// SIMATIC S7-200 project (STEP 7-Micro/WIN), CPU 226 REL 02.01

SYMBOL_TABLE 用户定义1
TS_IndexMotor    V1001.0
TS_ResetButton   V1000.0
Station_Alarm    V107.6
S6_Alarm         V168.7
S5_Alarm         V158.7
S4_Alarm         V148.7
S3_Alarm         V138.7
HomeApprop       M5.7
WaitStart        V3101.0
Running          V3101.1
Initilizing      V3100.1
WaitIni          V3100.0
TS_Rset_3D_0     V2000.7
TS_Rset_3C_0     V2000.5
TS_Rset_3B0      V2000.3
E_Stop           M0.0
Start_Button     M0.1
Stop_Button      M0.2
Reset_Button     M0.3
Bypass           M0.4
Safety_Relay     M0.5
MW_Switch        M0.6
Safety_Curtain   M0.7
S1_Ball_Screw    M1.0
S1_OE1           M1.1
S1_OE2           M1.2
S1_OE3           M1.3
S1_Cover_Group   M1.4
S1_Color         M1.5
S1_ORing         M1.6
SpareM1_7        M1.7
S2Ball_Screw     M2.0
S2OE21           M2.1
S2OE2            M2.2
S2OE3            M2.3
S2_Cover_Group   M2.4
Color_Sensor     M2.5
S2ORing          M2.6
Cyl3A_S0         M3.0
Cyl3A_S1         M3.1
Cyl3B_S0         M3.2
Cyl3B_S1         M3.3
Cy3C_S1          M3.5
Cyl3C_S0         M3.4
Cyl3D_S0         M3.6
CyL3D_S1         M3.7
Cyl_4A_S0        M4.0
Cyl4A_S1         M4.1
Cyl4B_S0         M4.2
Cyl4B_S1         M4.3
Cyl4C_S0         M4.4
Cyl4C_S1         M4.5
Cyl4D_S0         M4.6
Cyl4D_S1         M4.7
Laser_Marking    M5.0
Laser_done       M5.1
Cyl6A_S0         M6.0
Cyl6A_S1         M6.1
Cyl6B_S0         M6.2
Cyl6B_S1         M6.3
Cyl6C_S0         M6.4
Cyl6C_S1         M6.5
SpareM6_6        M6.6
SpareM6_7        M6.7
ServoMotorBLimit M7.0
Servo_Home_Pos   M7.1
ServoMotorFLimit M7.2
ServoAlarm       M7.3
ServoReady       M7.4
Cyl3E_S0         M8.0
Cyl3E_S1         M8.1
Cyl3F_S0         M8.2
Cyl3F_S1         M8.3
SpareM8_4        M8.4
SpareM8_5        M8.5
Cyl2A_S0         M8.6
Cyl2A_S1         M8.7
IndexOrig_Pos    M9.0
Reject_Box_1     M9.1
Reject_Box_2     M9.2
Reject_Box_3     M9.3
Reject_Box_4     M9.4
PC_Test_Complete_1 M9.5
PC_Test_Complete_2 M9.6
SafetyDoor       M9.7
CurrentTestOK_1  M10.0
CurrentTestNG_1  M10.1
RunTimeTestOK_1  M10.2
RunTimeTestNG_1  M10.3
LeakageTestOK_1  M10.4
LeakageTestNG_1  M10.5
LeakageTestAlarm_1 M10.6
Add_10N_Force_1  M10.7
CurrentTestOK_2  M11.0
CurrentTestNG_2  M11.1
RunTimeTestOK_2  M11.2
RunTimeTestNG_2  M11.3
LeakageTestOK_2  M11.4
LeakageTestNG_2  M11.5
LeakageTestAlarm_2 M11.6
Add_10N_Force_2  M11.7
CW               M20.0
CCW              M20.1
ServoEnable      M20.2
DelServoAlarm    M20.3
Up_Down_Cyl_1    M20.4
Up_Down_Cyl_2    M20.5
Pic_Product_Cyl_1 M20.6
Pic_Product_Cyl_2 M20.7
TW_G             M21.0
TW_R             M21.1
TW_Buzzer        M21.2
Reset_lamp       M21.3
Bypass_Lamp      M21.4
SV_3E_0          M22.0
SV_3E_1          M22.1
SV_3F_0          M22.2
SV_3F_1          M22.3
EnableTest_to_PC1 M22.4
EnableTest_to_PC2 M22.5
SV_3A_0          M23.0
SV_3A_1          M23.1
SV_3B_0          M23.2
SV_3B_1          M23.3
SV_3C_0          M23.4
SV_3C_1          M23.5
SV_3D_0          M23.6
SV_3D_1          M23.7
SV_4A_0          M24.0
SV_4A_1          M24.1
SV_4B_2mmCYL     M24.2
SV_4C_RotateCyl  M24.3
SV_4D_RotateCyl  M24.4
Index_Brake      M24.5
Servo_Brake      M24.6
MainValve        M24.7
Index_Motor      M25.0
ConverMotor      M25.1
RejectBox_Cyl    M25.2
Start_Laser      M25.3
Stop_Laser       M25.4
SpareM25_5       M25.5
Alarm1_ToPC      M25.6
Alarm2_ToPC      M25.7
StartLeakage_1   M26.0
ResetLeakage_1   M26.1
Romote_Eable_1   M26.2
StartLeakage_2   M27.0
ResetLeakage_2   M27.1
Romote_Eable_2   M27.2
StationRunTag    V0.0
TurnplateRunTag  V0.1
SysIniOk         V0.5
DeviceIniOk      V0.6
Ini_OK_Tag       V0.7
StationIniStatus V1.0
Station1IniStatus V1.1
Station2IniStatus V1.2
Station3IniStatus V1.3
Station4IniStatus V1.4
Station5IniStatus V1.5
Station6IniStatus V1.6
IniTags          V1.7
TypeCheckOk      V2.1
Auto_Mode        V3.0
TW_Ini_Status    V4.0
S5_To_S6_Ok      V9.0
S4_To_S5_Ok      V9.1
S3_To_S4_Ok      V9.2
S2_To_S3_Ok      V9.3
SS_Transfer_Ok   V9.7
Start_Signal     V10.7
S2_Complete_Tag  V27.7
下行汽缸AB           V36.1
通电汽缸             V36.2
移除砝码             V36.6
移除插座             V36.7
释放产品             V37.0
S3_CompleteTag   V37.7
S4_Product_Enable_Tag_1 V40.1
S4_Product_Enable_Tag_2 V40.2
S4_ProductEnable V40.3
S4_Complete_Tag  V47.7
Sent_Ok          V50.7
S5_Complete_Tag  V57.7
Release1st_1     V60.4
Release1st_2     V60.5
S6_Complete_Tag  V67.7
Fatal_Alarm      V107.7
TS_Start         V1000.1
TS_Stop          V1000.2
TS_Reset         V1000.3
Index_Signal_Edge V1000.7
Product_set      V1999.7
TS_Set_3A        V2000.0
TS_Reset_3A      V2000.1
TS_Set_3B        V2000.2
TS_Set_3C        V2000.4
TS_Set_3D        V2000.6
TS_Set_3E        V2001.0
TS_Set_3F        V2001.2
TS_Current_Test  V2001.4
TS_Set_4A        V2004.0
TS_Reset_4A      V2004.1
Maintain_mode    V2009.7
Single_Mode      V2019.7
TS_Laser_Test    V2049.0
TS_Laser_Stop    V2049.1
END_SYMBOL_TABLE

SYMBOL_TABLE S7-200 符号
Always_On        SM0.0    // 始终接通为 ON
First_Scan_On    SM0.1    // 仅第一个扫描周期中接通为 ON
Clock_1s         SM0.5    // 在 1 秒钟的循环周期内，接通为 ON 0.5 秒，关断为 OFF 0.5  秒
PLS0_Enable      SM67.7   // PTO0/PWM0 使能：1 = 使能
PLS1_Enable      SM77.7   // PTO1/PWM1 使能：1 = 使能
PLS0_Ctrl        SMB67    // PTO0/PMW0 监控，用于 Q0.0 上的 PTO（脉冲串输出）和PWM（脉冲宽度调制）
PLS1_Ctrl        SMB77    // PTO1/PWM1 监控，用于 Q0.1 上的 PTO（脉冲串输出）和 PWM（脉冲宽度调制）
PTO0_PC          SMD72    // PTO0 脉冲计数值：双字整数（1至2^32 - 1）
PTO1_PC          SMD82    // PTO1 脉冲计数值：双字整数（1至2^32 - 1）
PLS0_Cycle       SMW68    // PTO0/PWM0 周期时间值：字数据类型（2 至 65,535 个时基单位）
PLS1_Cycle       SMW78    // PTO1/PWM1 周期时间值：字数据类型（2 至 65,535 个时基单位）
END_SYMBOL_TABLE

ORGANIZATION_BLOCK Main_program:OB1
TITLE=项目信息 
// 这个PLC程序控制一个6工位转盘系统，用于在汽车零部件装配线上实现自动化装配和测试，主要针对刹车阀或油泵等部件。
// 系统通过PLC管理转盘的旋转和各工位的操作，支持自动和手动模式，并在自动模式下通过运行标志V0.0置位启动转盘运行。
// 程序记录测试结果和生产数据VW2050、VW2054，用于后续生产管理和质量控制。
// 物理设备包括6工位转盘、进料机构、类型检测机构、电气测试机构、泄漏测试机构、打标机构、下料机构、传感器和执行器。
// 
// 系统流程
// 操作员通过触摸屏通信监控系统状态，并可选择自动模式或手动模式运行。按下启动按钮后，若安全条件满足，系统将置位转盘运行标志，启动转盘旋转，各工位按序执行任务。系统上电时，系统初始化确保所有硬件复位并加载参数，设备初始化完成和系统初始化完成信号确认后，生产才能开始。
// 生产流程从上料工位控制开始，零件被放置在转盘上，通过传感器检测零件到位后，上料动作完成。转盘旋转到下一工位后，类型检测工位控制通过传感器识别刹车阀型号。随后，电气测试工位控制检测电气性能，合格与否记录在生产计数器中。接着，泄漏测试工位控制检查气密性，若泄漏测试仪报警触发，系统会停止该工位操作以防止次品流出。合格零件进入打标工位控制，由激光设备刻印标识，最后通过下料工位控制卸载成品，伺服马达控制将零件送至指定位置。
// 系统在运行过程中，急停按钮用于监控设备状态，确保异常时及时干预。急停按钮被按下时，系统会立即停止所有操作，包括复位转盘运行标志，确保紧急情况下设备停机。当安全门打开时，系统将阻止转盘运行标志的置位，确保人员安全。安全继电器断电时，系统直接切断转盘电机的电源，避免电气故障。气压开关检测到气压不足时，系统暂停所有气动执行器的操作，确保动作可靠。运行中若安全光栅被遮挡，系统不置位转盘旋转标志，保护操作员安全。伺服马达报警触发时，系统禁用伺服马达使能，防止设备损坏。转盘运行标志置位前，系统需确认安全门关闭、安全继电器正常、气压充足等条件，确保运行平稳。报警处理检测到异常时，系统根据报警类型停止相关工位操作，保障安全。
// 
// 
// 【代码最后更新与2008年6月10日】
BEGIN
Network 1 // 网络标题
// 网络注释
LD     Always_On:SM0.0
CALL   Station1_Load:SBR0
?000
Network 2
LD     Always_On:SM0.0
CALL   Station2_TypeCheck:SBR1
Network 3
LD     Auto_Mode:V3.0
AN     Single_Mode:V2019.7
O      V2010.3
AN     TS_ResetButton:V1000.0
AN     Reset_Button:M0.3
AN     TS_Stop:V1000.2
CALL   Station3_E_Test:SBR2
Network 4
LD     Auto_Mode:V3.0
AN     Single_Mode:V2019.7
O      V2010.4
AN     Reset_Button:M0.3
AN     TS_ResetButton:V1000.0
AN     TS_Stop:V1000.2
CALL   Station4_L_Test:SBR3
Network 5
LDN    Single_Mode:V2019.7
O      V2010.5
AN     TS_ResetButton:V1000.0
AN     Reset_Button:M0.3
AN     TS_Stop:V1000.2
CALL   Station5_LMark:SBR4
Network 6
LD     Auto_Mode:V3.0
AN     Single_Mode:V2019.7
O      V2010.6
AN     Reset_Button:M0.3
AN     TS_ResetButton:V1000.0
AN     TS_Stop:V1000.2
CALL   Station6_Unload:SBR5
Network 7
LD     Always_On:SM0.0
CALL   Machine_alarm:SBR6
Network 8
LD     Always_On:SM0.0
CALL   Product_alarm:SBR7
Network 9
LD     Always_On:SM0.0
CALL   Ini:SBR8
Network 10
LD     Always_On:SM0.0
CALL   Turn:SBR9
Network 11
LD     Always_On:SM0.0
CALL   Servo_motor:SBR10
Network 12
LD     Always_On:SM0.0
CALL   Input:SBR11
Network 13
LD     Always_On:SM0.0
CALL   Output:SBR12
Network 14
LD     Always_On:SM0.0
CALL   TP170:SBR13
Network 15
LD     Always_On:SM0.0
CALL   Tags:SBR14
Network 16
LD     Always_On:SM0.0
CALL   PowerOn:SBR15
Network 17
LD     Always_On:SM0.0
CALL   SyS_MSG:SBR16
Network 18
LD     Always_On:SM0.0
CALL   Man_MSG:SBR17
Network 19
LD     Always_On:SM0.0
CALL   Communication_Laser:SBR18
END_ORGANIZATION_BLOCK

SUBROUTINE_BLOCK Station1_Load:SBR0
TITLE=子程序注释
BEGIN
Network 1 // 网络标题
// 网络注释
LD     Safety_Curtain:M0.7
EU
=      Start_Signal:V10.7
END_SUBROUTINE_BLOCK

SUBROUTINE_BLOCK Station2_TypeCheck:SBR1
TITLE=子程序注释
BEGIN
Network 1
// 等待启动信号
LD     IndexOrig_Pos:M9.0
EU
A      SysIniOk:V0.5
A      V26.0
A      Auto_Mode:V3.0
AN     TS_ResetButton:V1000.0
MOVB   2, VB26
Network 2
// 固定产品
LDN    TurnplateRunTag:V0.1
A      V26.1
AN     Cyl2A_S0:M8.6
A      Cyl2A_S1:M8.7
LPS
A      T33
MOVB   4, VB26
LPP
TON    T33, +50
Network 3
LDN    TurnplateRunTag:V0.1
A      V26.2
AN     Cyl2A_S1:M8.7
A      Cyl2A_S0:M8.6
MOVB   8, VB26
Network 4
// vb=6,Type=007 878-04
LDN    TurnplateRunTag:V0.1
LD     V26.3
O      Maintain_mode:V2009.7
ALD
CALL   TypeCheck:SBR19
CALL   TypeCheck1:SBR20
Network 5
LDN    TurnplateRunTag:V0.1
A      V26.3
LPS
A      T35
MOVB   16, VB26
LPP
TON    T35, +50
Network 6
// 放开产品
LDN    TurnplateRunTag:V0.1
A      V26.4
A      Cyl2A_S0:M8.6
AN     Cyl2A_S1:M8.7
MOVB   32, VB26
Network 7
LDN    TurnplateRunTag:V0.1
A      V26.5
MOVB   1, VB26
Network 8
LDB=   VB21, VB23
OB=    VB21, 0
LDB=   VB22, VB23
OB=    VB22, 0
ALD
=      TypeCheckOk:V2.1
Network 9
LDB=   VB23, 0
=      V121.6
Network 10
LDB=   VB23, 5
OB=    VB23, 6
=      M21.6
Network 11
LDB=   VB23, 1
OB=    VB23, 3
OB=    VB23, 5
=      M26.6
Network 12
LDB=   VB23, 2
OB=    VB23, 3
OB=    VB23, 6
=      M26.7
Network 13
LDB=   VB23, 4
OB=    VB23, 5
OB=    VB23, 6
=      M27.6
END_SUBROUTINE_BLOCK

SUBROUTINE_BLOCK Station3_E_Test:SBR2
TITLE=vb30--3b39;T130-----T149
BEGIN
Network 1
// 等待启动信号
LD     IndexOrig_Pos:M9.0
EU
LPS
A      V30.3
A      SysIniOk:V0.5
A      V36.0
MOVB   2, VB36
LRD
AN     V30.1
MOVB   VB31, VB33
LPP
AN     V30.2
MOVB   VB32, VB34
Network 2
// v31.1汽缸A和B下行（对应m3.1和m3.3感应信号）
LDN    TurnplateRunTag:V0.1
A      V30.3
A      下行汽缸AB:V36.1
LPS
LDN    Cyl3A_S0:M3.0
A      Cyl3A_S1:M3.1
ON     V30.1
LDN    Cyl3B_S0:M3.2
A      Cyl3B_S1:M3.3
ON     V30.2
ALD
ALD
MOVB   4, VB36
LPP
TON    T131, +20
Network 3
// V36.2 给产品通电。汽缸E为水平方向方的通电汽缸,对应产品类型为1、2、3、4；
// 汽缸F为垂直方向的通电汽缸；对应产品类型为5、6
LDN    TurnplateRunTag:V0.1
A      V30.3
A      通电汽缸:V36.2
LPS
LDB<=  VB23, 4
AN     Cyl3F_S0:M8.2
A      Cyl3F_S1:M8.3
LDB>=  VB23, 5
AN     Cyl3E_S0:M8.0
A      Cyl3E_S1:M8.1
OLD
ALD
TON    T32, +0
A      T32
MOVB   8, VB36
LPP
TON    T132, +20
Network 4 // 网络标题
// v36.3为提供给PC的测试Ready 信号，m10.7,m11.7 电流测试完成信号(也即加砝码信号，PC提供)，v36.4加砝码
LDN    TurnplateRunTag:V0.1
A      V30.3
A      V36.3
LPS
LD     EnableTest_to_PC1:M22.4
A      Add_10N_Force_1:M10.7
ON     V30.1
O      CurrentTestNG_1:M10.1
LD     EnableTest_to_PC2:M22.5
A      Add_10N_Force_2:M11.7
ON     V30.2
O      CurrentTestNG_2:M11.1
ALD
ALD
MOVB   16, VB36
LPP
TON    T133, +1000
Network 5
// v36.5 砝码已加信号
LDN    TurnplateRunTag:V0.1
A      V30.3
A      V36.4
LPS
LDN    Cyl3C_S0:M3.4
ON     V30.1
O      CurrentTestNG_1:M10.1
LDN    Cyl3D_S0:M3.6
ON     V30.2
O      CurrentTestNG_2:M11.1
ALD
ALD
TON    T34, +100
A      T34
MOVB   32, VB36
LPP
TON    T134, +40
Network 6
// 测试完成信号
LDN    TurnplateRunTag:V0.1
A      V30.3
A      V36.5
LPS
LD     PC_Test_Complete_1:M9.5
ON     V30.1
LD     PC_Test_Complete_2:M9.6
ON     V30.2
ALD
ALD
MOVB   64, VB36
LPP
TON    T135, +300
Network 7
// 去除砝码信号
LDN    TurnplateRunTag:V0.1
A      V30.3
A      移除砝码:V36.6
LPS
A      Cyl3C_S0:M3.4
A      Cyl3D_S0:M3.6
MOVB   128, VB36
LPP
TON    T136, +20
Network 8
// 断开通电插座
LDN    TurnplateRunTag:V0.1
A      V30.3
A      移除插座:V36.7
LPS
A      Cyl3E_S0:M8.0
A      Cyl3F_S0:M8.2
AN     Cyl3E_S1:M8.1
AN     Cyl3F_S1:M8.3
MOVB   1, VB37
AENO
MOVB   0, VB36
LPP
TON    T137, +20
Network 9
// 释放产品
LDN    TurnplateRunTag:V0.1
A      V30.3
A      释放产品:V37.0
LPS
A      Cyl3A_S0:M3.0
A      Cyl3B_S0:M3.2
AN     Cyl3A_S1:M3.1
AN     Cyl3B_S1:M3.3
MOVB   2, VB37
LPP
TON    T138, +20
Network 10
// 确定产品状态,v37.7=工作完成标志
LDN    TurnplateRunTag:V0.1
A      V30.3
A      V37.1
LPS
A      CurrentTestOK_1:M10.0
A      RunTimeTestOK_1:M10.2
AN     CurrentTestNG_1:M10.1
AN     RunTimeTestNG_1:M10.3
MOVB   31, VB33
AENO
=      L63.7
LRD
A      CurrentTestOK_1:M10.0
A      RunTimeTestNG_1:M10.3
MOVB   22, VB33
AENO
O      L63.7
=      L63.6
LRD
A      CurrentTestNG_1:M10.1
MOVB   21, VB33
AENO
O      L63.6
=      L63.5
LRD
A      V30.4
O      L63.5
=      L63.4
LRD
AN     V30.1
O      L63.4
LPS
A      CurrentTestOK_2:M11.0
A      RunTimeTestOK_2:M11.2
AN     CurrentTestNG_2:M11.1
AN     RunTimeTestNG_2:M11.3
MOVB   31, VB34
AENO
=      L63.3
LRD
A      CurrentTestOK_2:M11.0
A      RunTimeTestNG_2:M11.3
MOVB   22, VB34
AENO
O      L63.3
=      L63.2
LRD
A      CurrentTestNG_2:M11.1
MOVB   21, VB34
AENO
O      L63.2
=      L63.1
LRD
A      V30.5
O      L63.1
=      L63.0
LPP
AN     V30.2
O      L63.0
MOVB   128, VB37
LPP
TON    T139, +20
Network 11
LDN    TurnplateRunTag:V0.1
AN     TurnplateRunTag:V0.1
A      V30.3
A      S3_CompleteTag:V37.7
AN     EnableTest_to_PC1:M22.4
AN     EnableTest_to_PC2:M22.5
MOVB   1, VB36
AENO
MOVB   0, VB37
END_SUBROUTINE_BLOCK

SUBROUTINE_BLOCK Station4_L_Test:SBR3
TITLE=vb40--3b49;T150----T169
BEGIN
Network 1
// 等待启动
LD     IndexOrig_Pos:M9.0
EU
LPS
A      S4_ProductEnable:V40.3
A      SysIniOk:V0.5
A      V46.0
MOVB   2, VB46
LRD
AN     S4_ProductEnable:V40.3
LPS
A      S4_Product_Enable_Tag_1:V40.1
MOVB   32, VB43
LPP
A      S4_Product_Enable_Tag_2:V40.2
MOVB   32, VB44
LPP
LPS
AN     S4_Product_Enable_Tag_1:V40.1
MOVB   VB41, VB43
LPP
AN     S4_Product_Enable_Tag_2:V40.2
MOVB   VB42, VB44
Network 2
// v46.1汽缸A下行
LD     S4_ProductEnable:V40.3
A      V46.1
LPS
A      Cyl4A_S1:M4.1
AN     Cyl_4A_S0:M4.0
MOVB   4, VB46
LPP
TON    T151, +20
Network 3
// 汽缸C/D锁定
LD     S4_ProductEnable:V40.3
A      V46.2
LPS
LDN    Cyl4C_S0:M4.4
A      Cyl4C_S1:M4.5
ON     S4_Product_Enable_Tag_1:V40.1
LDN    Cyl4D_S0:M4.6
A      Cyl4D_S1:M4.7
ON     S4_Product_Enable_Tag_2:V40.2
ALD
ALD
MOVB   8, VB46
LPP
TON    T152, +20
Network 4 // 网络标题
// 汽缸B上行
LD     S4_ProductEnable:V40.3
A      V46.3
LPS
A      Cyl4B_S0:M4.2
AN     Cyl4B_S1:M4.3
MOVB   16, VB46
LPP
TON    T153, +20
Network 5
// 等待测试结果
LD     S4_ProductEnable:V40.3
A      V46.4
LPS
A      LeakageTestOK_1:M10.4
AN     LeakageTestNG_1:M10.5
AN     LeakageTestAlarm_1:M10.6
MOVB   32, VB43
AENO
=      L63.7
LRD
LD     LeakageTestNG_1:M10.5
O      LeakageTestAlarm_1:M10.6
ALD
MOVB   23, VB43
AENO
MOVB   0, VB47
AENO
O      L63.7
=      L63.6
LRD
AN     S4_Product_Enable_Tag_1:V40.1
O      L63.6
LPS
A      LeakageTestOK_2:M11.4
AN     LeakageTestNG_2:M11.5
AN     LeakageTestAlarm_2:M11.6
MOVB   32, VB44
AENO
=      L63.5
LRD
LD     LeakageTestNG_2:M11.5
O      LeakageTestAlarm_2:M11.6
ALD
MOVB   23, VB44
AENO
MOVB   0, VB47
AENO
O      L63.5
=      L63.4
LPP
AN     S4_Product_Enable_Tag_2:V40.2
O      L63.4
MOVB   32, VB46
LPP
TON    T154, +150
Network 6
// 汽缸
LD     S4_ProductEnable:V40.3
A      V46.5
LPS
A      Cyl4C_S0:M4.4
A      Cyl4D_S0:M4.6
AN     Cyl4C_S1:M4.5
AN     Cyl4D_S1:M4.7
MOVB   64, VB46
LPP
TON    T155, +20
Network 7
LD     S4_ProductEnable:V40.3
A      V46.6
LPS
A      Cyl4B_S1:M4.3
AN     Cyl4B_S0:M4.2
MOVB   128, VB46
LPP
TON    T156, +20
Network 8
LD     S4_ProductEnable:V40.3
A      V46.7
LPS
A      Cyl_4A_S0:M4.0
AN     Cyl4A_S1:M4.1
MOVB   1, VB47
AENO
A      V47.0
MOVB   0, VB46
LPP
TON    T157, +50
Network 9
// 释放产品
LD     S4_ProductEnable:V40.3
A      V47.0
LPS
A      Cyl_4A_S0:M4.0
MOVB   2, VB47
LPP
TON    T158, +20
Network 10
// 确定产品状态,v47.7=工作完成标志
LD     S4_ProductEnable:V40.3
A      V47.1
MOVB   128, VB47
TON    T159, +20
Network 11
LDN    StationRunTag:V0.0
AN     TurnplateRunTag:V0.1
A      S4_ProductEnable:V40.3
LPS
A      S4_Complete_Tag:V47.7
MOVB   1, VB46
AENO
MOVB   0, VB47
LPP
TON    T160, +20
Network 14 // 网络标题
// 网络注释
END_SUBROUTINE_BLOCK

SUBROUTINE_BLOCK Station5_LMark:SBR4
TITLE=VB50---VB59;  T170-----T179
BEGIN
Network 1
// 等待启动
LD     IndexOrig_Pos:M9.0
EU
LPS
A      V50.3
A      SysIniOk:V0.5
A      V56.0
MOVB   2, VB56
LRD
AN     V50.1
MOVB   VB51, VB53
LPP
AN     V50.2
MOVB   VB52, VB54
Network 2
// 启动打标
LDN    TurnplateRunTag:V0.1
A      V50.3
A      V56.1
LD     Q6.5
A      V50.1
LD     Q7.5
A      V50.2
OLD
ALD
MOVB   4, VB56
Network 3
// 等待打标完成
LDN    TurnplateRunTag:V0.1
A      V50.3
A      V56.2
LPS
A      Laser_done:M5.1
ED
MOVB   8, VB56
LRD
TON    T201, +250
LPP
R      Sent_Ok:V50.7, 1
Network 4
// 传送工位结果
LDN    TurnplateRunTag:V0.1
A      V50.3
A      V56.3
LPS
A      V50.1
MOVB   34, VB53
AENO
=      L63.7
LPP
A      V50.2
MOVB   34, VB54
AENO
O      L63.7
LDB=   VB53, 34
ON     V50.1
ALD
LDB=   VB54, 34
ON     V50.2
ALD
MOVB   1, VB56
Network 5 // 网络标题
// 网络注释
END_SUBROUTINE_BLOCK

SUBROUTINE_BLOCK Station6_Unload:SBR5
TITLE=VB60----VB69;    T180--T199
BEGIN
Network 1
LDN    Index_Motor:M25.0
AN     TurnplateRunTag:V0.1
O      V2006.4
O      V2006.5
O      V2006.6
O      V2006.7
O      V66.4
A      Cyl6A_S0:M6.0
=      ServoEnable:M20.2
=      Servo_Brake:M24.6
Network 2
// 到达放料位置后清除 产品代码；设定下一个目标位置
LD     V60.6
LPS
A      M31.1
AN     M31.2
AN     M31.3
AN     M31.4
LPS
LDB=   VB61, 22
OB=    VB62, 22
ALD
MOVD   +7500, VD268
LRD
LDB=   VB61, 23
OB=    VB62, 23
ALD
MOVD   +16000, VD272
LRD
LDB=   VB61, 29
OB=    VB62, 29
ALD
MOVD   +24500, VD276
LPP
LDB=   VB61, 34
OB=    VB62, 34
ALD
MOVD   +32800, VD260
LRD
A      M31.2
AN     M31.3
AN     M31.4
LPS
LDB=   VB61, 23
OB=    VB62, 23
ALD
MOVD   +7500, VD272
LRD
LDB=   VB61, 29
OB=    VB62, 29
ALD
MOVD   +16000, VD276
LPP
LDB=   VB61, 34
OB=    VB62, 34
ALD
MOVD   +24300, VD260
LRD
A      M31.3
AN     M31.4
LPS
LDB=   VB61, 29
OB=    VB62, 29
ALD
MOVD   +7500, VD276
LPP
LDB=   VB61, 34
OB=    VB62, 34
ALD
MOVD   +16300, VD260
LPP
A      M31.4
LDB=   VB61, 34
OB=    VB62, 34
ALD
MOVD   +7800, VD260
Network 3
LD     V60.6
AN     V1002.1
AN     V1002.2
AW<>   VW61, +0
A      V66.6
MOVB   0, VB61
AENO
MOVB   0, VB62
Network 4
LDN    Always_On:SM0.0
A      V60.6
LPS
A      M31.3
LDB=   VB61, 34
OB=    VB62, 34
ALD
MOVD   +16500, VD260
LPP
A      M31.4
LDB=   VB61, 34
OB=    VB62, 34
ALD
MOVD   +8000, VD260
Network 5 // 网络标题
// 等待启动
LD     IndexOrig_Pos:M9.0
EU
A      SysIniOk:V0.5
A      V60.3
A      V66.0
MOVB   2, VB66
Network 6
// 汽缸A下行
LDN    TurnplateRunTag:V0.1
A      V60.3
A      V66.1
LPS
A      Cyl6A_S1:M6.1
AN     Cyl6A_S0:M6.0
MOVB   4, VB66
LRD
TON    T181, +80
LRD
EU
AB<>   VB61, 34
A      V60.1
+I     +1, VW2054
LRD
EU
AB<>   VB62, 34
A      V60.2
+I     +1, VW2054
LRD
EU
AB=    VB61, 34
A      V60.1
+I     +1, VW2050
LPP
EU
AB=    VB62, 34
A      V60.2
+I     +1, VW2050
Network 7
LD     Always_On:SM0.0
MOVW   VW2050, VW2058
+I     VW2054, VW2058
Network 8
// 汽缸BC取料
LDN    TurnplateRunTag:V0.1
A      V60.3
A      V66.2
LPS
LDN    Cyl6B_S0:M6.2
A      Cyl6B_S1:M6.3
ON     V60.1
LDN    Cyl6C_S0:M6.4
A      Cyl6C_S1:M6.5
ON     V60.2
ALD
ALD
MOVB   8, VB66
LPP
TON    T182, +80
Network 9
// 汽缸A上行
LDN    TurnplateRunTag:V0.1
A      V60.3
A      V66.3
LPS
A      V360.1
MOVD   +44300, VD260
AENO
AD=    VD260, +44300
=      L63.7
LRD
A      V360.2
MOVD   +10500, VD264
AENO
AD=    VD264, +10500
O      L63.7
=      L63.6
LRD
A      V360.3
MOVD   +19000, VD268
AENO
AD=    VD268, +19000
O      L63.6
=      L63.5
LRD
A      V360.4
MOVD   +27500, VD272
AENO
AD=    VD272, +27500
O      L63.5
=      L63.4
LRD
A      V360.5
MOVD   +36000, VD276
AENO
AD=    VD276, +36000
O      L63.4
A      Cyl6A_S0:M6.0
MOVB   16, VB66
LPP
TON    T183, +50
Network 10
// 马达定位完成信号V60.6
LDN    TurnplateRunTag:V0.1
A      V60.3
A      V66.4
LPS
LD     V360.1
LD     M31.5
O      M5.6
ALD
LD     V360.2
A      M31.1
LD     V360.3
A      M31.2
OLD
LD     V360.4
A      M31.3
OLD
LD     V360.5
A      M31.4
OLD
OLD
ALD
LPS
A      T204
MOVB   64, VB66
LPP
TON    T204, +5
LPP
TON    T184, +150
Network 11
// 汽缸A下行
LDN    TurnplateRunTag:V0.1
A      V60.3
A      V66.5
LPS
A      Cyl6A_S1:M6.1
AN     Cyl6A_S0:M6.0
MOVB   64, VB66
LPP
TON    T185, +80
Network 12
// 释放产品的判断条件待加V60.4\V60.5\（根据测试结果的优先级别）
LDN    TurnplateRunTag:V0.1
A      V66.6
LPS
A      Cyl6B_S0:M6.2
A      V1002.1
MOVB   0, VB61
AENO
=      L63.7
LRD
A      V1002.2
O      L63.7
LPS
A      Cyl6C_S0:M6.4
A      V1002.2
MOVB   0, VB62
AENO
=      L63.6
LPP
A      V1002.1
O      L63.6
=      L63.5
LPP
AN     V1002.1
AN     V1002.2
A      Cyl6B_S0:M6.2
MOVB   0, VB61
AENO
A      Cyl6C_S0:M6.4
MOVB   0, VB62
AENO
O      L63.5
LD     M31.1
A      Reject_Box_1:M9.1
LD     M31.2
A      Reject_Box_2:M9.2
OLD
LD     M31.3
A      Reject_Box_3:M9.3
OLD
LD     M31.4
A      Reject_Box_4:M9.4
OLD
O      M31.5
O      M5.6
ALD
MOVB   128, VB66
Network 13
// 放料监控
LDN    TurnplateRunTag:V0.1
A      V66.6
TON    T186, +100
Network 14
LD     M5.6
R      PLS0_Enable:SM67.7, 1
PLS    0
Network 15
// 汽缸A上行,mb31=0清除马达定位完成信号
LDN    TurnplateRunTag:V0.1
A      V66.7
LPS
A      Cyl6A_S0:M6.0
AN     Cyl6A_S1:M6.1
MOVB   1, VB67
AENO
MOVB   0, VB66
LRD
R      V1002.1, 2
LPP
TON    T187, +80
Network 16
// 根据条件判断是继续放料还是回到原始位置。该条件待加
LDN    TurnplateRunTag:V0.1
A      V67.0
LPS
AW=    VW61, +0
A      Servo_Home_Pos:M7.1
MOVB   1, VB66
AENO
MOVB   0, MB31
AENO
A      V66.0
MOVB   0, VB67
LPP
AW<>   VW61, +0
MOVB   16, VB66
AENO
A      V66.4
MOVB   0, VB67
END_SUBROUTINE_BLOCK

SUBROUTINE_BLOCK Machine_alarm:SBR6
TITLE=
BEGIN
Network 1 // 网络标题
// 急停被按下
LD     E_Stop:M0.0
=      V106.0
Network 2
// 安全门被打开
LDN    SafetyDoor:M9.7
O      V106.1
AN     TS_Reset:V1000.3
AN     TS_ResetButton:V1000.0
AN     Reset_Button:M0.3
=      V106.1
Network 3
// 安全继电器断电
LDN    Safety_Relay:M0.5
O      V106.1
AN     TS_Reset:V1000.3
AN     TS_ResetButton:V1000.0
AN     Reset_Button:M0.3
=      V106.2
Network 4
// 气压低
LDN    MW_Switch:M0.6
O      V106.3
AN     TS_Reset:V1000.3
AN     TS_ResetButton:V1000.0
AN     Reset_Button:M0.3
=      V106.3
Network 5
// 运行中安全光栅被遮挡
LD     TurnplateRunTag:V0.1
AN     Safety_Curtain:M0.7
O      V106.4
AN     TS_Reset:V1000.3
AN     TS_ResetButton:V1000.0
AN     Reset_Button:M0.3
=      V106.4
Network 6
// 饲服马达报警
LD     ServoAlarm:M7.3
O      V106.5
AN     TS_Reset:V1000.3
AN     Always_On:SM0.0
AN     TS_ResetButton:V1000.0
AN     Reset_Button:M0.3
=      V106.5
Network 7
// 泄露测试仪报警-1
LD     LeakageTestAlarm_1:M10.6
O      V106.6
AN     TS_Reset:V1000.3
AN     Always_On:SM0.0
AN     TS_ResetButton:V1000.0
AN     Reset_Button:M0.3
=      V106.6
Network 8
// 泄露测试仪报警-2
LD     LeakageTestAlarm_2:M11.6
O      V106.7
AN     TS_Reset:V1000.3
AN     Always_On:SM0.0
AN     TS_ResetButton:V1000.0
AN     Reset_Button:M0.3
=      V106.7
Network 9
LDW<>  VW61, +0
A      ServoMotorBLimit:M7.0
O      V107.0
AN     TS_ResetButton:V1000.0
AN     Always_On:SM0.0
AN     Reset_Button:M0.3
=      V107.0
Network 10
LDW<>  VW61, +0
A      ServoMotorFLimit:M7.2
O      V107.1
AN     TS_ResetButton:V1000.0
AN     Always_On:SM0.0
AN     Reset_Button:M0.3
=      V107.1
Network 11
// 停机报警（运行时单工位报警不影响其他工位运行，待运行结束后停机）
LDN    V106.0
AN     V106.1
AN     V106.2
AN     V106.3
AN     V106.4
AN     V106.5
AN     V106.6
AN     V106.7
AN     V107.0
AN     V107.1
AN     V107.2
AN     V107.3
AN     V107.4
AN     V107.5
LDN    Station_Alarm:V107.6
O      StationRunTag:V0.0
ALD
=      Fatal_Alarm:V107.7
Network 12
// 电测试工位汽缸A下行失败--取料
LD     T131
AN     Cyl3A_S1:M3.1
O      V136.0
AN     TS_Reset:V1000.3
AN     TS_ResetButton:V1000.0
AN     Reset_Button:M0.3
=      V136.0
Network 13
// 电测试工位汽缸B下行失败--取料
LD     T131
AN     Cyl3B_S1:M3.3
O      V136.1
AN     TS_Reset:V1000.3
AN     TS_ResetButton:V1000.0
AN     Reset_Button:M0.3
=      V136.1
Network 14
// 电测试工位通电汽缸E前进失败--取料
LD     T132
AB>=   VB23, 5
AN     Cyl3E_S1:M8.1
O      V136.2
AN     TS_Reset:V1000.3
AN     TS_ResetButton:V1000.0
AN     Reset_Button:M0.3
=      V136.2
Network 15
// 电测试工位通电汽缸F前进失败--
LD     T132
AB<=   VB23, 4
AN     Cyl3F_S1:M8.3
O      V136.3
AN     TS_Reset:V1000.3
AN     TS_ResetButton:V1000.0
AN     Reset_Button:M0.3
=      V136.3
Network 16
// 电测试工位PC发送加10N1信号超时--
LD     T133
A      V30.1
AN     Add_10N_Force_1:M10.7
O      V136.4
AN     TS_Reset:V1000.3
AN     TS_ResetButton:V1000.0
AN     Reset_Button:M0.3
=      V136.4
Network 17
// 电测试工位PC发送加10N2信号超时--
LD     T133
A      V30.2
AN     Add_10N_Force_2:M11.7
O      V136.5
AN     TS_Reset:V1000.3
AN     TS_ResetButton:V1000.0
AN     Reset_Button:M0.3
=      V136.5
Network 18
// 电测试工位加10N汽缸1下行失败
LD     T134
A      V30.1
A      Cyl3C_S0:M3.4
O      V136.6
AN     TS_Reset:V1000.3
AN     TS_ResetButton:V1000.0
AN     Reset_Button:M0.3
=      V136.6
Network 19
// 电测试工位加10N汽缸2下行失败
LD     T134
A      V30.2
A      Cyl3D_S0:M3.6
O      V136.7
AN     TS_Reset:V1000.3
AN     TS_ResetButton:V1000.0
AN     Reset_Button:M0.3
=      V136.7
Network 20
// 电测试工位PC发送完成信号1超时
LD     T135
A      V30.1
AN     PC_Test_Complete_1:M9.5
O      V137.0
AN     TS_Reset:V1000.3
AN     TS_ResetButton:V1000.0
AN     Reset_Button:M0.3
=      V137.0
Network 21
// 电测试工位PC发送完成信号2超时
LD     T135
A      V30.2
AN     PC_Test_Complete_2:M9.6
O      V137.1
AN     TS_Reset:V1000.3
AN     TS_ResetButton:V1000.0
AN     Reset_Button:M0.3
=      V137.1
Network 22
// 电测试工位 加10N汽缸1上行失败
LD     T136
O      T191
AN     Cyl3C_S0:M3.4
O      V137.2
AN     TS_Reset:V1000.3
AN     TS_ResetButton:V1000.0
AN     Reset_Button:M0.3
=      V137.2
Network 23
// 电测试工位 加10N汽缸上行失败
LD     T136
O      T191
AN     Cyl3D_S0:M3.6
O      V137.3
AN     TS_Reset:V1000.3
AN     TS_ResetButton:V1000.0
AN     Reset_Button:M0.3
=      V137.3
Network 24
// 电测试工位通电汽缸1后退失败
LD     T137
O      T190
AN     Cyl3E_S0:M8.0
O      V137.4
AN     TS_Reset:V1000.3
AN     TS_ResetButton:V1000.0
AN     Reset_Button:M0.3
=      V137.4
Network 25
// 电测试工位 通电汽缸汽缸2下行失败
LD     T137
O      T190
AN     Cyl3F_S0:M8.2
O      V137.5
AN     TS_Reset:V1000.3
AN     TS_ResetButton:V1000.0
AN     Reset_Button:M0.3
=      V137.5
Network 26
// 电测试工位 汽缸A上行失败
LD     T138
O      T192
AN     Cyl3A_S0:M3.0
O      V137.6
AN     TS_Reset:V1000.3
AN     TS_ResetButton:V1000.0
AN     Reset_Button:M0.3
=      V137.6
Network 27
// 电测试工位 汽缸B上行失败
LD     T138
O      T192
AN     Cyl3B_S0:M3.2
O      V137.7
AN     TS_Reset:V1000.3
AN     TS_ResetButton:V1000.0
AN     Reset_Button:M0.3
=      V137.7
Network 28
// 电测试工位 测试结果未知
LD     T139
O      V138.0
AN     TS_Reset:V1000.3
AN     TS_ResetButton:V1000.0
AN     Reset_Button:M0.3
=      V138.0
Network 29
// 泄露测试工位 汽缸A下行失败
LD     T151
O      V146.0
AN     TS_Reset:V1000.3
AN     TS_ResetButton:V1000.0
AN     Reset_Button:M0.3
=      V146.0
Network 30
// 泄露测试工位 锁定汽缸B上行失败
LD     T153
O      V146.1
AN     TS_Reset:V1000.3
AN     TS_ResetButton:V1000.0
AN     Reset_Button:M0.3
=      V146.1
Network 31
// 泄露测试工位 锁定汽缸C前进失败
LD     T152
A      S4_Product_Enable_Tag_1:V40.1
AN     Cyl4C_S1:M4.5
O      V146.2
AN     TS_Reset:V1000.3
AN     TS_ResetButton:V1000.0
AN     Reset_Button:M0.3
=      V146.2
Network 32
// 泄露测试工位 锁定汽缸D前进失败
LD     T152
A      S4_Product_Enable_Tag_2:V40.2
AN     Cyl4D_S1:M4.7
O      V146.3
AN     TS_Reset:V1000.3
AN     TS_ResetButton:V1000.0
AN     Reset_Button:M0.3
=      V146.3
Network 33
// 测试结果未知
LD     T154
O      V146.4
AN     TS_Reset:V1000.3
AN     TS_ResetButton:V1000.0
AN     Reset_Button:M0.3
=      V146.4
Network 34
// 汽缸C后退失败
LD     T155
O      T194
AN     Cyl4C_S1:M4.5
O      V146.5
AN     TS_Reset:V1000.3
AN     TS_ResetButton:V1000.0
AN     Reset_Button:M0.3
=      V146.5
Network 35
// 汽缸D后退失败
LD     T155
O      T194
AN     Cyl4D_S1:M4.7
O      V146.6
AN     TS_Reset:V1000.3
AN     TS_ResetButton:V1000.0
AN     Reset_Button:M0.3
=      V146.6
Network 36
// 汽缸B上行失败
LD     T156
O      T193
O      V146.7
AN     TS_Reset:V1000.3
AN     TS_ResetButton:V1000.0
AN     Reset_Button:M0.3
=      V146.7
Network 37
// 汽缸A上行失败
LD     T157
O      T195
O      V147.0
AN     TS_Reset:V1000.3
AN     TS_ResetButton:V1000.0
AN     Reset_Button:M0.3
=      V147.0
Network 38
// 字符错误
LDW<>  VW2020, +0
AW=    VW2022, +0
O      V156.0
AN     TS_ResetButton:V1000.0
AN     Reset_Button:M0.3
=      V156.0
Network 39
// 系统错误，如通讯
LD     T201
O      V156.1
AN     TS_ResetButton:V1000.0
AN     Reset_Button:M0.3
=      V156.1
Network 40
// 软件错误
LDW<>  VW2020, +0
AW=    VW2022, +3
O      V156.2
AN     TS_ResetButton:V1000.0
AN     Reset_Button:M0.3
=      V156.2
Network 41
// 汽缸A下行失败
LD     T181
O      T185
O      V166.0
AN     TS_Reset:V1000.3
AN     TS_ResetButton:V1000.0
AN     Reset_Button:M0.3
=      V166.0
Network 42
// 汽缸B抓产品失败
LD     T182
A      V60.1
AN     Cyl6B_S1:M6.3
O      V166.1
AN     TS_Reset:V1000.3
AN     TS_ResetButton:V1000.0
AN     Reset_Button:M0.3
=      V166.1
Network 43
// 汽缸C抓产品失败
LD     T182
A      V60.2
AN     Cyl6C_S1:M6.5
O      V166.2
AN     TS_Reset:V1000.3
AN     TS_ResetButton:V1000.0
AN     Reset_Button:M0.3
=      V166.2
Network 44
// 汽缸A上行失败
LD     T183
O      T187
O      T197
O      V166.3
AN     TS_Reset:V1000.3
AN     Always_On:SM0.0
AN     TS_ResetButton:V1000.0
AN     Reset_Button:M0.3
=      V166.3
Network 45
// 马达定位超时
LD     T184
O      V166.4
AN     TS_Reset:V1000.3
AN     TS_ResetButton:V1000.0
AN     Reset_Button:M0.3
=      V166.4
Network 46
// 汽缸B放料失败
LD     T186
A      V1002.1
O      V166.5
AN     TS_Reset:V1000.3
AN     TS_ResetButton:V1000.0
AN     Reset_Button:M0.3
=      V166.5
Network 47
// 汽缸C放料失败
LD     T186
A      V1002.2
O      V166.6
AN     TS_Reset:V1000.3
AN     TS_ResetButton:V1000.0
AN     Reset_Button:M0.3
=      V166.6
Network 48
LDB<>  VB136, 0
OB<>   VB137, 0
O      V138.0
ON     Fatal_Alarm:V107.7
O      S3_Alarm:V138.7
AN     TS_Reset:V1000.3
AN     TS_ResetButton:V1000.0
AN     Reset_Button:M0.3
LPS
=      S3_Alarm:V138.7
MOVD   +0, VD36
A      V30.1
AB<>   VB33, 21
AB<>   VB33, 22
MOVB   29, VB33
LPP
A      V30.2
AB<>   VB34, 21
AB<>   VB34, 22
MOVB   29, VB34
Network 49
LDB<>  VB146, 0
OB<>   VB147, 0
ON     Fatal_Alarm:V107.7
O      S4_Alarm:V148.7
AN     TS_Reset:V1000.3
AN     TS_ResetButton:V1000.0
AN     Reset_Button:M0.3
LPS
=      S4_Alarm:V148.7
MOVW   +0, VW46
A      S4_Product_Enable_Tag_1:V40.1
AB<=   VB23, 4
AB<>   VB41, 21
AB<>   VB41, 22
AB<>   VB43, 21
AB<>   VB43, 22
AB<>   VB43, 23
MOVB   29, VB43
LPP
A      S4_Product_Enable_Tag_2:V40.2
AB<=   VB23, 4
AB<>   VB42, 21
AB<>   VB42, 22
AB<>   VB44, 21
AB<>   VB44, 22
AB<>   VB44, 23
MOVB   29, VB44
Network 50
LD     V156.1
ON     Fatal_Alarm:V107.7
O      S5_Alarm:V158.7
AN     TS_Reset:V1000.3
AN     TS_ResetButton:V1000.0
AN     Reset_Button:M0.3
LPS
=      S5_Alarm:V158.7
MOVW   +0, VW56
A      V50.1
AB<>   VB51, 21
AB<>   VB51, 21
AB<>   VB53, 21
AB<>   VB53, 22
AB<>   VB53, 23
AB<>   VB53, 34
MOVB   29, VB53
LPP
A      V50.2
AB<>   VB52, 21
AB<>   VB52, 21
AB<>   VB54, 21
AB<>   VB54, 22
AB<>   VB54, 23
AB<>   VB54, 34
MOVB   29, VB54
Network 51
LDB<>  VB166, 0
OB<>   VB167, 0
O      S6_Alarm:V168.7
ON     Fatal_Alarm:V107.7
AN     TS_Reset:V1000.3
AN     TS_ResetButton:V1000.0
AN     Reset_Button:M0.3
=      S6_Alarm:V168.7
MOVW   +0, VW66
Network 52
// 汽缸等的报警
LD     S3_Alarm:V138.7
O      S4_Alarm:V148.7
O      S5_Alarm:V158.7
O      S6_Alarm:V168.7
O      Station_Alarm:V107.6
AN     TS_ResetButton:V1000.0
=      Station_Alarm:V107.6
END_SUBROUTINE_BLOCK

SUBROUTINE_BLOCK Product_alarm:SBR7
TITLE=
BEGIN
Network 1 // 网络标题
// 类型不一致报警1
LD     StationRunTag:V0.0
AN     TurnplateRunTag:V0.1
AB<>   VB21, VB23
O      V121.0
AN     TypeCheckOk:V2.1
AN     Reset_Button:M0.3
AN     Always_On:SM0.0
AN     TS_ResetButton:V1000.0
=      V121.0
Network 2 // 网络标题
// 类型不一致报警2
LD     StationRunTag:V0.0
AN     TurnplateRunTag:V0.1
AB<>   VB22, VB23
O      V121.1
AN     TypeCheckOk:V2.1
AN     Always_On:SM0.0
AN     Reset_Button:M0.3
AN     TS_ResetButton:V1000.0
=      V121.1
Network 3 // 网络标题
// 缺少密封圈报警1
LD     StationRunTag:V0.0
AN     TurnplateRunTag:V0.1
AB<>   VB21, 0
AN     S1_ORing:M1.6
O      V121.2
AN     TypeCheckOk:V2.1
AN     Always_On:SM0.0
AN     Reset_Button:M0.3
AN     TS_ResetButton:V1000.0
=      V121.2
Network 4 // 网络标题
// 缺少密封圈报警2
LD     StationRunTag:V0.0
AN     TurnplateRunTag:V0.1
AB<>   VB22, 0
AN     S2ORing:M2.6
O      V121.3
AN     TypeCheckOk:V2.1
AN     Always_On:SM0.0
AN     Reset_Button:M0.3
AN     TS_ResetButton:V1000.0
=      V121.3
Network 5 // 网络标题
// 缺少BallScrew报警1
LD     StationRunTag:V0.0
AN     TurnplateRunTag:V0.1
AB<>   VB21, 0
AN     S1_Ball_Screw:M1.0
O      V121.4
AN     TypeCheckOk:V2.1
AN     Always_On:SM0.0
AN     Reset_Button:M0.3
AN     TS_ResetButton:V1000.0
=      V121.4
Network 6 // 网络标题
// 缺少BallScrew报警2
LD     StationRunTag:V0.0
AN     TurnplateRunTag:V0.1
AB<>   VB22, 0
AN     S2Ball_Screw:M2.0
O      V121.5
AN     TypeCheckOk:V2.1
AN     Always_On:SM0.0
AN     Reset_Button:M0.3
AN     TS_ResetButton:V1000.0
=      V121.5
Network 7
LDB=   VB23, 0
=      V121.6
Network 8 // 网络标题
// 电流测试NG提示
LD     StationRunTag:V0.0
AN     TurnplateRunTag:V0.1
A      CurrentTestNG_1:M10.1
O      V122.0
AN     TypeCheckOk:V2.1
AN     Always_On:SM0.0
AN     Reset_Button:M0.3
AN     TS_ResetButton:V1000.0
=      V122.0
Network 9 // 网络标题
// 电流测试NG提示
LD     StationRunTag:V0.0
AN     TurnplateRunTag:V0.1
A      CurrentTestNG_2:M11.1
O      V122.1
AN     TypeCheckOk:V2.1
AN     Always_On:SM0.0
AN     Reset_Button:M0.3
AN     TS_ResetButton:V1000.0
=      V122.1
Network 10 // 网络标题
// 跑合测试NG提示1
LD     StationRunTag:V0.0
AN     TurnplateRunTag:V0.1
A      RunTimeTestNG_1:M10.3
O      V122.2
AN     TypeCheckOk:V2.1
AN     Always_On:SM0.0
AN     Reset_Button:M0.3
AN     TS_ResetButton:V1000.0
=      V122.2
Network 11 // 网络标题
// 跑合测试NG提示2
LD     StationRunTag:V0.0
AN     TurnplateRunTag:V0.1
A      RunTimeTestNG_2:M11.3
O      V122.3
AN     TypeCheckOk:V2.1
AN     Always_On:SM0.0
AN     Reset_Button:M0.3
AN     TS_ResetButton:V1000.0
=      V122.3
Network 12 // 网络标题
// 泄露测试NG提示1
LD     StationRunTag:V0.0
AN     TurnplateRunTag:V0.1
A      LeakageTestNG_1:M10.5
O      V122.4
AN     TypeCheckOk:V2.1
AN     Always_On:SM0.0
AN     Reset_Button:M0.3
AN     TS_ResetButton:V1000.0
=      V122.4
Network 13 // 网络标题
// 泄露测试NG提示1
LD     StationRunTag:V0.0
AN     TurnplateRunTag:V0.1
A      LeakageTestNG_2:M11.5
O      V122.5
AN     TypeCheckOk:V2.1
AN     Always_On:SM0.0
AN     Reset_Button:M0.3
AN     TS_ResetButton:V1000.0
=      V122.5
Network 14
LDB<>  VB121, 0
OB<>   VB122, 0
=      V122.7
Network 15
LD     V66.6
A      Reject_Box_1:M9.1
EU
INCB   VB91
Network 16
LD     V66.6
A      Reject_Box_2:M9.2
EU
INCB   VB92
Network 17
LD     V66.6
A      Reject_Box_3:M9.3
EU
INCB   VB93
Network 18
LD     V66.6
A      Reject_Box_1:M9.1
EU
INCB   VB94
Network 19
// 电流测试不合格箱满
LD     Servo_Home_Pos:M7.1
A      Reject_Box_1:M9.1
OB=    VB91, 15
O      V123.1
AN     TS_ResetButton:V1000.0
AN     TS_Reset:V1000.3
AN     Reset_Button:M0.3
=      V123.1
MOVB   0, VB91
Network 20
// 跑合测试不合格箱满
LD     Servo_Home_Pos:M7.1
A      Reject_Box_2:M9.2
OB=    VB92, 15
O      V123.2
AN     TS_ResetButton:V1000.0
AN     TS_Reset:V1000.3
AN     Reset_Button:M0.3
=      V123.2
MOVB   0, VB92
Network 21
// 泄露测试不合格箱满
LD     Servo_Home_Pos:M7.1
A      Reject_Box_3:M9.3
OB=    VB93, 15
O      V123.3
AN     TS_ResetButton:V1000.0
AN     TS_Reset:V1000.3
AN     Reset_Button:M0.3
=      V123.3
MOVB   0, VB93
Network 22
// 未测试箱满
LD     Servo_Home_Pos:M7.1
A      Reject_Box_4:M9.4
OB=    VB94, 15
O      V123.4
AN     TS_ResetButton:V1000.0
AN     TS_Reset:V1000.3
AN     Reset_Button:M0.3
=      V123.4
MOVB   0, VB94
Network 23
LD     V123.1
O      V123.2
O      V123.3
O      V123.4
=      V123.7
Network 24
LD     Always_On:SM0.0
MOVB   VB123, VB3123
END_SUBROUTINE_BLOCK

SUBROUTINE_BLOCK Ini:SBR8
TITLE=
BEGIN
Network 1 // 网络标题
// 网络注释
LD     First_Scan_On:SM0.1
O      TW_Ini_Status:V4.0
AN     Reset_Button:M0.3
AN     TS_ResetButton:V1000.0
AN     TS_Reset:V1000.3
=      TW_Ini_Status:V4.0
Network 2
// vw2020=0,vw2022=4清除打标机报警信息
LD     TS_ResetButton:V1000.0
LPS
MOVB   1, VB39
AENO
MOVB   1, VB49
AENO
MOVB   1, VB59
AENO
MOVB   1, VB69
LRD
MOVW   +0, VW2020
AENO
MOVW   +4, VW2022
LRD
S      Auto_Mode:V3.0, 1
LPP
R      Index_Signal_Edge:V1000.7, 1
Network 3
LD     DeviceIniOk:V0.6
MOVB   0, VB39
AENO
MOVB   0, VB49
AENO
MOVB   0, VB59
AENO
MOVB   0, VB69
Network 4
LD     V39.0
LPS
A      Cyl3E_S0:M8.0
A      Cyl3F_S0:M8.2
MOVB   2, VB39
LPP
TON    T190, +50
Network 5
LD     V39.1
LPS
A      Cyl3C_S0:M3.4
A      Cyl3D_S0:M3.6
MOVB   4, VB39
LPP
TON    T191, +50
Network 6
LD     V39.2
LPS
A      Cyl3A_S0:M3.0
A      Cyl3B_S0:M3.2
MOVB   8, VB39
LPP
TON    T192, +50
Network 7
LD     V39.2
A      Cyl3A_S0:M3.0
A      Cyl3B_S0:M3.2
A      Cyl3C_S0:M3.4
A      Cyl3D_S0:M3.6
A      Cyl3E_S0:M8.0
A      Cyl3F_S0:M8.2
MOVB   0, VB39
Network 8
LD     V49.0
LPS
A      Cyl4B_S1:M4.3
MOVB   2, VB49
LPP
TON    T193, +50
Network 9
LD     V49.1
LPS
A      Cyl4C_S0:M4.4
A      Cyl4D_S0:M4.6
MOVB   4, VB49
LPP
TON    T194, +50
Network 10
LD     V49.2
LPS
A      Cyl_4A_S0:M4.0
MOVB   8, VB49
LPP
TON    T195, +50
Network 11
LD     V49.3
A      Cyl_4A_S0:M4.0
A      Cyl4B_S0:M4.2
A      Cyl4C_S0:M4.4
A      Cyl4D_S0:M4.6
MOVB   0, VB49
Network 12
LD     V69.0
LPS
A      Cyl6B_S0:M6.2
A      Cyl6C_S0:M6.4
MOVB   2, VB69
LPP
TON    T196, +50
Network 13
LD     V69.1
LPS
A      Cyl6A_S0:M6.0
MOVB   4, VB69
LPP
TON    T197, +50
Network 14
// 准备找原点
LD     V69.2
LPS
A      Servo_Home_Pos:M7.1
MOVB   8, VB69
LPP
AN     Servo_Home_Pos:M7.1
MOVB   16, VB69
Network 15
// CCW方向运行一段距离
LD     V69.3
AN     Servo_Home_Pos:M7.1
A      M31.6
MOVB   16, VB69
Network 16
// CW方向找原点
LD     V69.4
A      Servo_Home_Pos:M7.1
MOVB   32, VB69
Network 17
// CW方向找原点
LD     V69.5
R      M31.6, 2
AN     M31.6
AN     M31.7
MOVB   64, VB69
Network 18
// CW方向找原点
LD     V69.6
MOVB   0, VB69
Network 19
LD     WaitIni:V3100.0
AN     Cyl2A_S0:M8.6
=      V126.0
Network 20
LD     WaitIni:V3100.0
AN     Cyl3A_S0:M3.0
=      V126.1
Network 21
LD     WaitIni:V3100.0
AN     Cyl3B_S0:M3.2
=      V126.2
Network 22
LD     WaitIni:V3100.0
AN     Cyl3C_S0:M3.4
=      V126.3
Network 23
LD     WaitIni:V3100.0
AN     Cyl3D_S0:M3.6
=      V126.4
Network 24
LD     WaitIni:V3100.0
AN     Cyl3E_S0:M8.0
=      V126.5
Network 25
LD     WaitIni:V3100.0
AN     Cyl3F_S0:M8.2
=      V126.6
Network 26
LD     WaitIni:V3100.0
AN     Cyl_4A_S0:M4.0
=      V126.7
Network 27
LD     WaitIni:V3100.0
AN     Cyl4B_S1:M4.3
=      V125.0
Network 28
LD     WaitIni:V3100.0
AN     Cyl4C_S0:M4.4
=      V125.1
Network 29
LD     WaitIni:V3100.0
AN     Cyl4D_S0:M4.6
=      V125.2
Network 30
LD     WaitIni:V3100.0
AN     Servo_Home_Pos:M7.1
=      V125.3
Network 31
LD     WaitIni:V3100.0
AN     Cyl6A_S0:M6.0
=      V125.4
Network 32
LD     WaitIni:V3100.0
AN     Cyl6B_S0:M6.2
=      V125.5
Network 33
LD     WaitIni:V3100.0
AN     Cyl6C_S0:M6.4
=      V125.6
Network 34
LD     WaitIni:V3100.0
AN     IndexOrig_Pos:M9.0
=      V125.7
END_SUBROUTINE_BLOCK

SUBROUTINE_BLOCK Turn:SBR9
TITLE=vb9
BEGIN
Network 1
// 传送类型检测结果
LD     TurnplateRunTag:V0.1
A      Index_Motor:M25.0
AN     StationRunTag:V0.0
LPS
EU
MOVB   VB53, VB61
AENO
MOVB   VB54, VB62
AENO
AB=    VB53, VB61
AB=    VB54, VB62
=      S5_To_S6_Ok:V9.0
LRD
A      S5_To_S6_Ok:V9.0
EU
MOVB   VB43, VB51
AENO
MOVB   VB44, VB52
AENO
AB=    VB43, VB51
AB=    VB44, VB52
=      S4_To_S5_Ok:V9.1
LRD
A      S4_To_S5_Ok:V9.1
EU
MOVB   VB33, VB41
AENO
MOVB   VB34, VB42
AENO
AB=    VB33, VB41
AB=    VB34, VB42
=      S3_To_S4_Ok:V9.2
LPP
A      S3_To_S4_Ok:V9.2
EU
LPS
LDB=   VB21, VB23
OB=    VB21, 0
ALD
MOVB   VB21, VB31
AENO
AB=    VB21, VB31
=      L63.7
LPP
AB<>   VB21, VB23
AB<>   VB21, 0
MOVB   29, VB31
AENO
AB=    29, VB31
O      L63.7
LPS
LDB=   VB22, VB23
OB=    VB22, 0
ALD
MOVB   VB22, VB32
AENO
AB=    VB22, VB32
=      L63.6
LPP
AB<>   VB22, VB23
AB<>   VB22, 0
MOVB   29, VB32
AENO
AB=    29, VB32
O      L63.6
=      S2_To_S3_Ok:V9.3
Network 2
LD     S5_To_S6_Ok:V9.0
A      S4_To_S5_Ok:V9.1
A      S3_To_S4_Ok:V9.2
A      S2_To_S3_Ok:V9.3
=      SS_Transfer_Ok:V9.7
Network 3
LDN    Station_Alarm:V107.6
A      Fatal_Alarm:V107.7
AN     StationRunTag:V0.0
O      TS_IndexMotor:V1001.0
A      Index_Motor:M25.0
=      TurnplateRunTag:V0.1
Network 4
LDN    TS_ResetButton:V1000.0
A      SysIniOk:V0.5
A      Safety_Curtain:M0.7
O      TS_IndexMotor:V1001.0
EU
O      TS_ResetButton:V1000.0
S      Index_Brake:M24.5, 1
Network 5
LD     IndexOrig_Pos:M9.0
O      Station_Alarm:V107.6
O      StationRunTag:V0.0
ON     Fatal_Alarm:V107.7
EU
AN     TS_ResetButton:V1000.0
R      Index_Brake:M24.5, 1
Network 6
LD     Always_On:SM0.0
=      MainValve:M24.7
Network 7
LD     TurnplateRunTag:V0.1
MOVD   +0, VD2000
AENO
MOVW   +0, VW2005
Network 8
LD     Safety_Curtain:M0.7
EU
LD     StationRunTag:V0.0
O      WaitStart:V3101.0
ALD
S      V3.7, 1
Network 9
LD     IndexOrig_Pos:M9.0
EU
R      V3.7, 1
END_SUBROUTINE_BLOCK

SUBROUTINE_BLOCK Servo_motor:SBR10
TITLE=料箱位置：OK     VD260      Current NG VD264    RunTime  VD268     Leakage NG VD270   ;No Test :VD 274
// 
BEGIN
Network 1
LD     V66.7
O      TS_ResetButton:V1000.0
O      First_Scan_On:SM0.1
A      M31.0
R      M31.0, 1
Network 2
LD     V66.7
O      TS_ResetButton:V1000.0
O      First_Scan_On:SM0.1
A      M31.1
R      M31.1, 1
Network 3
LD     V66.7
O      TS_ResetButton:V1000.0
O      First_Scan_On:SM0.1
A      M31.2
R      M31.2, 1
Network 4
LD     V66.7
O      TS_ResetButton:V1000.0
O      First_Scan_On:SM0.1
A      M31.3
R      M31.3, 1
Network 5
LD     V66.7
O      TS_ResetButton:V1000.0
O      First_Scan_On:SM0.1
A      M31.4
R      M31.4, 1
Network 6
LD     V66.7
O      TS_ResetButton:V1000.0
O      First_Scan_On:SM0.1
A      M31.5
R      M31.5, 1
Network 7
LD     V69.5
O      TS_ResetButton:V1000.0
O      First_Scan_On:SM0.1
A      M31.6
R      M31.6, 1
Network 8
LD     V69.5
O      TS_ResetButton:V1000.0
O      First_Scan_On:SM0.1
A      M31.7
R      M31.7, 1
Network 9
// OK成品，放入OK区(最外面的)  45000/500=90R
LD     V66.4
A      V360.1
A      V60.3
EU
MOVB   16#85, PLS0_Ctrl:SMB67
MOVW   +80, PLS0_Cycle:SMW68
MOVD   VD260, PTO0_PC:SMD72
PLS    0
ATCH   OK_Pos:INT5, 19
ENI
Network 10
// Current废品，放入第1个料箱（最里面的）
LD     V66.4
A      V360.2
A      V60.3
EU
MOVB   16#85, PLS0_Ctrl:SMB67
MOVW   +80, PLS0_Cycle:SMW68
MOVD   VD264, PTO0_PC:SMD72
PLS    0
ATCH   Current_NG:INT1, 19
ENI
Network 11
// RunTime 废品，放入第2料箱
LD     V66.4
A      V360.3
A      V60.3
EU
MOVB   16#85, PLS0_Ctrl:SMB67
MOVW   +80, PLS0_Cycle:SMW68
MOVD   VD268, PTO0_PC:SMD72
PLS    0
ATCH   RunTime_NG:INT2, 19
ENI
Network 12
// Leakage  废品，放入第3个料箱
LD     V66.4
A      V360.4
A      V60.3
EU
MOVB   16#85, PLS0_Ctrl:SMB67
MOVW   +80, PLS0_Cycle:SMW68
MOVD   VD272, PTO0_PC:SMD72
PLS    0
ATCH   LKG_NG:INT3, 19
ENI
Network 13
// 未测，放入第4个料箱
LD     V66.4
A      V360.5
A      V60.3
EU
MOVB   16#85, PLS0_Ctrl:SMB67
MOVW   +80, PLS0_Cycle:SMW68
MOVD   VD276, PTO0_PC:SMD72
PLS    0
ATCH   NoTest:INT4, 19
ENI
Network 14
// 返回原始位置（取料位置）
LD     V67.0
AW=    VW61, +0
O      TS_ResetButton:V1000.0
LPS
AN     Servo_Home_Pos:M7.1
MOVB   16#85, PLS1_Ctrl:SMB77
MOVW   +80, PLS1_Cycle:SMW78
MOVD   +100, PTO1_PC:SMD82
PLS    1
ATCH   Orig_Pos:INT0, 20
ENI
LPP
A      Servo_Home_Pos:M7.1
R      PLS1_Enable:SM77.7, 1
R      V2007.0, 1
PLS    1
Network 15
// CW方向寻找原点（取料位置）
LD     V69.4
O      V2007.0
LPS
AN     Servo_Home_Pos:M7.1
MOVB   16#85, PLS1_Ctrl:SMB77
MOVW   +80, PLS1_Cycle:SMW78
MOVD   +100, PTO1_PC:SMD82
PLS    1
ATCH   Servo_Ini:INT6, 20
ENI
LPP
A      Servo_Home_Pos:M7.1
R      PLS1_Enable:SM77.7, 1
R      V2007.0, 1
PLS    1
Network 16
// 如果原点信号有，先CCW方向运行一段距离
LD     V69.3
AN     Always_On:SM0.0
EU
MOVB   16#85, PLS0_Ctrl:SMB67
MOVW   +200, PLS0_Cycle:SMW68
MOVD   VD270, PTO0_PC:SMD72
PLS    0
ATCH   Servo_Ini:INT6, 19
ENI
Network 17
// 手动快速运行（CW方）
LD     V2006.4
AN     ServoMotorFLimit:M7.2
MOVB   16#85, PLS1_Ctrl:SMB77
MOVW   +100, PLS1_Cycle:SMW78
MOVD   +2000, PTO1_PC:SMD82
PLS    1
ATCH   None:INT7, 20
ENI
Network 18
// 手动慢速速运行（CW方）
LD     V2006.6
AN     ServoMotorFLimit:M7.2
MOVB   16#85, PLS1_Ctrl:SMB77
MOVW   +500, PLS1_Cycle:SMW78
MOVD   +2000, PTO1_PC:SMD82
PLS    1
ATCH   None:INT7, 20
ENI
Network 19
// 手动快速运行（CCW方向）
LD     V2006.5
AN     ServoMotorFLimit:M7.2
MOVB   16#85, PLS0_Ctrl:SMB67
MOVW   +100, PLS0_Cycle:SMW68
MOVD   +2000, PTO0_PC:SMD72
PLS    0
ATCH   None:INT7, 19
ENI
Network 20
// 手动慢速运行（CCW方向）
LD     V2006.7
AN     ServoMotorFLimit:M7.2
MOVB   16#85, PLS0_Ctrl:SMB67
MOVW   +500, PLS0_Cycle:SMW68
MOVD   +2000, PTO0_PC:SMD72
PLS    0
ATCH   None:INT7, 19
ENI
Network 21 // 网络标题
// 网络注释
END_SUBROUTINE_BLOCK

SUBROUTINE_BLOCK Input:SBR11
TITLE=
BEGIN
Network 1 // 网络标题
// 网络注释
LDN    I0.0
=      E_Stop:M0.0
Network 2
LD     I0.1
=      Start_Button:M0.1
Network 3
LD     I0.2
=      Stop_Button:M0.2
Network 4
LD     I0.3
=      Reset_Button:M0.3
Network 5
LD     I0.4
=      Bypass:M0.4
Network 6
LD     I0.5
=      Safety_Relay:M0.5
Network 7
LD     I0.6
=      MW_Switch:M0.6
Network 8
LD     I0.7
=      Safety_Curtain:M0.7
Network 9
LD     I1.0
=      S1_Ball_Screw:M1.0
Network 10
LD     I1.1
=      S1_OE1:M1.1
Network 11
LD     I1.2
=      S1_OE2:M1.2
Network 12
LD     I1.3
=      S1_OE3:M1.3
Network 13
LD     I1.4
=      S1_Cover_Group:M1.4
Network 14
LD     I1.5
=      S1_Color:M1.5
Network 15
LD     I1.6
=      S1_ORing:M1.6
Network 16
LD     I1.7
=      SpareM1_7:M1.7
Network 17
LD     I2.0
=      S2Ball_Screw:M2.0
Network 18
LD     I2.1
=      S2OE21:M2.1
Network 19
LD     I2.2
=      S2OE2:M2.2
Network 20
LD     I2.3
=      S2OE3:M2.3
Network 21
LD     I2.4
=      S2_Cover_Group:M2.4
Network 22
LD     I2.5
=      Color_Sensor:M2.5
Network 23
LD     I2.6
=      S2ORing:M2.6
Network 24
LD     I2.7
=      M2.7
Network 25
LD     I3.0
=      Cyl3A_S0:M3.0
Network 26
LD     I3.1
=      Cyl3A_S1:M3.1
Network 27
LD     I3.2
=      Cyl3B_S0:M3.2
Network 28
LD     I3.3
=      Cyl3B_S1:M3.3
Network 29
LD     I3.4
=      Cyl3C_S0:M3.4
Network 30
LD     I3.5
=      Cy3C_S1:M3.5
Network 31
LD     I3.6
=      Cyl3D_S0:M3.6
Network 32 // 			
LD     I3.7
=      CyL3D_S1:M3.7
Network 33
LD     I4.0
=      Cyl_4A_S0:M4.0
Network 34
LD     I4.1
=      Cyl4A_S1:M4.1
Network 35
LD     I4.2
=      Cyl4B_S0:M4.2
Network 36
LD     I4.3
=      Cyl4B_S1:M4.3
Network 37
LD     I4.4
=      Cyl4C_S0:M4.4
Network 38
LD     I4.5
=      Cyl4C_S1:M4.5
Network 39
LD     I4.6
=      Cyl4D_S0:M4.6
Network 40
LD     I4.7
=      Cyl4D_S1:M4.7
Network 41
LD     I5.0
=      Laser_Marking:M5.0
Network 42
LD     I5.1
=      Laser_done:M5.1
Network 43
LD     I5.2
=      M5.2
Network 44
LD     I5.3
=      M5.3
Network 45
LD     I5.4
=      M5.4
Network 46
LD     I5.5
=      M5.5
Network 47
LD     I5.6
=      M5.6
Network 48
LD     I6.0
=      Cyl6A_S0:M6.0
Network 49
LD     I6.1
=      Cyl6A_S1:M6.1
Network 50
LD     I6.3
=      Cyl6B_S0:M6.2
Network 51
LD     I6.2
=      Cyl6B_S1:M6.3
Network 52
LD     I6.5
=      Cyl6C_S0:M6.4
Network 53
LD     I6.4
=      Cyl6C_S1:M6.5
Network 54
LD     I6.6
=      SpareM6_6:M6.6
Network 55
LD     I6.7
=      SpareM6_7:M6.7
Network 56
LD     I5.4
=      ServoMotorBLimit:M7.0
Network 57
LD     I5.5
=      Servo_Home_Pos:M7.1
Network 58
LD     I5.7
=      ServoMotorFLimit:M7.2
Network 59
LD     I7.3
=      ServoAlarm:M7.3
Network 60
LD     I7.4
=      ServoReady:M7.4
Network 61
LD     I7.5
=      M7.5
Network 62
LD     I7.6
=      M7.6
Network 63
LD     I7.7
=      M7.7
Network 64
LD     I8.0
=      Cyl3E_S0:M8.0
Network 65
LD     I8.1
=      Cyl3E_S1:M8.1
Network 66
LD     I8.2
=      Cyl3F_S0:M8.2
Network 67
LD     I8.3
=      Cyl3F_S1:M8.3
Network 68
LD     I8.4
=      SpareM8_4:M8.4
Network 69
LD     I8.5
=      SpareM8_5:M8.5
Network 70
LD     I8.6
=      Cyl2A_S0:M8.6
Network 71
LD     I8.7
=      Cyl2A_S1:M8.7
Network 72
LD     I9.0
=      IndexOrig_Pos:M9.0
EU
S      Index_Signal_Edge:V1000.7, 1
Network 73
LD     I9.1
=      Reject_Box_1:M9.1
Network 74
LD     I9.2
=      Reject_Box_2:M9.2
Network 75
LD     I9.3
=      Reject_Box_3:M9.3
Network 76
LD     I9.4
=      Reject_Box_4:M9.4
Network 77
LD     I9.5
=      PC_Test_Complete_1:M9.5
Network 78
LD     I9.6
=      PC_Test_Complete_2:M9.6
Network 79
LD     I9.7
O      Bypass:M0.4
=      SafetyDoor:M9.7
Network 80
LD     I10.0
=      CurrentTestOK_1:M10.0
Network 81
LD     I10.1
=      CurrentTestNG_1:M10.1
Network 82
LD     I10.2
=      RunTimeTestOK_1:M10.2
Network 83
LD     I10.3
=      RunTimeTestNG_1:M10.3
Network 84
LD     I10.4
=      LeakageTestOK_1:M10.4
Network 85
LD     I10.5
=      LeakageTestNG_1:M10.5
Network 86
LD     I10.6
=      LeakageTestAlarm_1:M10.6
Network 87
LD     I10.7
=      Add_10N_Force_1:M10.7
Network 88
LD     I11.0
=      CurrentTestOK_2:M11.0
Network 89
LD     I11.1
=      CurrentTestNG_2:M11.1
Network 90
LD     I11.2
=      RunTimeTestOK_2:M11.2
Network 91
LD     I11.3
=      RunTimeTestNG_2:M11.3
Network 92
LD     I11.4
=      LeakageTestOK_2:M11.4
Network 93
LD     I11.5
=      LeakageTestNG_2:M11.5
Network 94
LD     I11.6
=      LeakageTestAlarm_2:M11.6
Network 95
LD     I11.7
=      Add_10N_Force_2:M11.7
END_SUBROUTINE_BLOCK

SUBROUTINE_BLOCK Output:SBR12
TITLE=
BEGIN
Network 2
// Q0.1 CCW
Network 3
LD     V26.1
O      M27.7
AN     TS_ResetButton:V1000.0
AN     Index_Motor:M25.0
A      IndexOrig_Pos:M9.0
AN     Reset_Button:M0.3
AN     V26.2
=      M27.7
Network 4
// 双控下行固定汽缸A
LD     释放产品:V37.0
O      Index_Motor:M25.0
O      V39.2
O      SV_3A_0:M23.0
O      Reset_Button:M0.3
O      TS_ResetButton:V1000.0
AN     下行汽缸AB:V36.1
=      SV_3A_0:M23.0
Network 5
// 双控下行固定汽缸A
LD     下行汽缸AB:V36.1
O      SV_3A_1:M23.1
AN     释放产品:V37.0
AN     Reset_Button:M0.3
AN     TS_ResetButton:V1000.0
AN     Index_Motor:M25.0
AN     S3_Alarm:V138.7
AN     V39.2
A      Fatal_Alarm:V107.7
A      IndexOrig_Pos:M9.0
A      V30.1
=      SV_3A_1:M23.1
Network 6
// 双控下行固定汽缸B
LD     释放产品:V37.0
O      V39.2
O      Index_Motor:M25.0
O      SV_3B_0:M23.2
O      Reset_Button:M0.3
O      TS_ResetButton:V1000.0
AN     下行汽缸AB:V36.1
=      SV_3B_0:M23.2
Network 7
// 双控下行固定汽缸B
LD     下行汽缸AB:V36.1
O      SV_3B_1:M23.3
AN     释放产品:V37.0
AN     Reset_Button:M0.3
AN     TS_ResetButton:V1000.0
AN     S3_Alarm:V138.7
AN     V39.2
A      Fatal_Alarm:V107.7
A      IndexOrig_Pos:M9.0
A      V30.2
=      SV_3B_1:M23.3
Network 8
// 通电汽缸
LD     通电汽缸:V36.2
O      SV_3E_1:M22.1
AN     移除插座:V36.7
AN     Index_Motor:M25.0
AN     TS_ResetButton:V1000.0
AN     S3_Alarm:V138.7
AN     Reset_Button:M0.3
A      Fatal_Alarm:V107.7
AN     V39.0
A      IndexOrig_Pos:M9.0
AB>    VB23, 4
=      SV_3E_1:M22.1
Network 9
// 通电汽缸
LD     通电汽缸:V36.2
O      SV_3F_1:M22.3
AN     移除插座:V36.7
AN     Index_Motor:M25.0
AN     TS_ResetButton:V1000.0
AN     S3_Alarm:V138.7
AN     Reset_Button:M0.3
A      Fatal_Alarm:V107.7
AN     V39.0
A      IndexOrig_Pos:M9.0
AB<=   VB23, 4
=      SV_3F_1:M22.3
Network 10
LD     V36.3
O      EnableTest_to_PC1:M22.4
AN     Index_Motor:M25.0
AN     S3_CompleteTag:V37.7
AN     S3_Alarm:V138.7
AN     V39.0
A      IndexOrig_Pos:M9.0
A      Fatal_Alarm:V107.7
A      V30.1
=      EnableTest_to_PC1:M22.4
Network 11
LD     V36.3
O      EnableTest_to_PC2:M22.5
AN     Index_Motor:M25.0
AN     S3_CompleteTag:V37.7
AN     S3_Alarm:V138.7
AN     V39.0
A      IndexOrig_Pos:M9.0
A      Fatal_Alarm:V107.7
A      V30.2
=      EnableTest_to_PC2:M22.5
Network 12
// 加砝码汽缸
LD     移除砝码:V36.6
O      V39.1
ON     IndexOrig_Pos:M9.0
O      V39.1
O      SV_3C_0:M23.4
O      TS_ResetButton:V1000.0
O      Reset_Button:M0.3
AN     V36.4
=      SV_3C_0:M23.4
Network 13
// 加砝码汽缸
LD     V36.4
A      Add_10N_Force_1:M10.7
O      SV_3C_1:M23.5
AN     Index_Motor:M25.0
AN     Reset_Button:M0.3
AN     S3_Alarm:V138.7
AN     TS_ResetButton:V1000.0
A      Fatal_Alarm:V107.7
AN     移除砝码:V36.6
AN     V39.1
A      IndexOrig_Pos:M9.0
A      V30.1
=      SV_3C_1:M23.5
Network 14
// 加砝码汽缸
LD     移除砝码:V36.6
O      V39.1
ON     IndexOrig_Pos:M9.0
O      SV_3D_0:M23.6
O      TS_ResetButton:V1000.0
O      Reset_Button:M0.3
AN     V36.4
=      SV_3D_0:M23.6
Network 15
// 加砝码汽缸
LD     V36.4
A      Add_10N_Force_2:M11.7
O      SV_3D_1:M23.7
AN     Index_Motor:M25.0
AN     Reset_Button:M0.3
AN     S3_Alarm:V138.7
AN     TS_ResetButton:V1000.0
A      Fatal_Alarm:V107.7
AN     移除砝码:V36.6
AN     V39.1
A      IndexOrig_Pos:M9.0
A      V30.2
=      SV_3D_1:M23.7
Network 16
// Run Time 使能信号
LD     V36.5
O      M22.6
O      M22.7
AN     Index_Motor:M25.0
AN     移除砝码:V36.6
AN     S3_Alarm:V138.7
A      Fatal_Alarm:V107.7
AN     V39.1
A      IndexOrig_Pos:M9.0
LPS
A      V30.1
A      Add_10N_Force_1:M10.7
=      M22.6
LPP
A      V30.2
A      Add_10N_Force_2:M11.7
=      M22.7
Network 17
// 泄露测试工位
LD     V46.7
O      Index_Motor:M25.0
O      V49.2
O      TS_ResetButton:V1000.0
O      Reset_Button:M0.3
O      SV_4A_0:M24.0
AN     V46.1
=      SV_4A_0:M24.0
Network 18
// 泄露测试工位
LD     V46.1
O      SV_4A_1:M24.1
AN     V46.7
AN     Reset_Button:M0.3
AN     S4_Alarm:V148.7
AN     TS_ResetButton:V1000.0
A      Fatal_Alarm:V107.7
AN     Index_Motor:M25.0
AN     V49.2
A      IndexOrig_Pos:M9.0
=      SV_4A_1:M24.1
Network 19
// 推进汽缸
LD     V46.6
O      V49.0
O      Reset_Button:M0.3
O      TS_ResetButton:V1000.0
O      SV_4B_2mmCYL:M24.2
AN     V46.3
=      SV_4B_2mmCYL:M24.2
Network 20
// 2mm提升汽缸1??
LD     V46.2
O      SV_4C_RotateCyl:M24.3
AN     V46.5
AN     S4_Alarm:V148.7
AN     Index_Motor:M25.0
AN     V49.1
A      Fatal_Alarm:V107.7
A      S4_Product_Enable_Tag_1:V40.1
A      IndexOrig_Pos:M9.0
=      SV_4C_RotateCyl:M24.3
Network 21
// 2mm提升汽缸2??
LD     V46.2
O      SV_4D_RotateCyl:M24.4
AN     V46.5
AN     S4_Alarm:V148.7
AN     Index_Motor:M25.0
A      Fatal_Alarm:V107.7
AN     V49.1
A      S4_Product_Enable_Tag_2:V40.2
A      IndexOrig_Pos:M9.0
=      SV_4D_RotateCyl:M24.4
Network 22
LD     Fatal_Alarm:V107.7
ON     Station_Alarm:V107.6
=      ConverMotor:M25.1
Network 23
LD     V46.4
A      S4_Product_Enable_Tag_1:V40.1
=      StartLeakage_1:M26.0
Network 24
LD     V46.4
A      S4_Product_Enable_Tag_2:V40.2
=      StartLeakage_2:M27.0
Network 25
LD     V46.5
O      V46.1
=      ResetLeakage_1:M26.1
Network 26
LD     V46.5
O      V46.1
=      ResetLeakage_2:M27.1
Network 27
// 启动打印信号是600ms的高电平脉冲信号
LD     V56.1
O      M26.5
AN     V56.0
AN     Index_Motor:M25.0
AN     T172
A      V50.1
A      V50.3
A      IndexOrig_Pos:M9.0
=      M26.5
TON    T172, +800
Network 28
// 启动打印信号是600ms的高电平脉冲信号
LD     V56.1
O      M27.5
AN     V56.0
AN     Index_Motor:M25.0
AN     T172
A      V50.2
A      V50.3
A      IndexOrig_Pos:M9.0
=      M27.5
TON    T172, +800
Network 29
LD     V66.3
O      V66.7
O      V69.1
O      Index_Motor:M25.0
O      Up_Down_Cyl_1:M20.4
AN     V66.5
AN     V66.1
O      TS_ResetButton:V1000.0
=      Up_Down_Cyl_1:M20.4
Network 30
LD     V66.1
O      V66.5
O      Up_Down_Cyl_2:M20.5
AN     V66.3
AN     Index_Motor:M25.0
AN     S6_Alarm:V168.7
AN     V66.7
A      Fatal_Alarm:V107.7
AN     V69.1
A      V60.3
A      IndexOrig_Pos:M9.0
=      Up_Down_Cyl_2:M20.5
Network 31
LD     V66.2
O      Pic_Product_Cyl_1:M20.6
LDN    V66.6
O      V1002.2
ALD
AN     V69.0
A      Fatal_Alarm:V107.7
AN     Index_Motor:M25.0
A      IndexOrig_Pos:M9.0
=      Pic_Product_Cyl_1:M20.6
Network 32
LD     V66.2
O      Pic_Product_Cyl_2:M20.7
LDN    V66.6
O      V1002.1
ALD
AN     V69.0
A      Fatal_Alarm:V107.7
AN     Index_Motor:M25.0
A      IndexOrig_Pos:M9.0
=      Pic_Product_Cyl_2:M20.7
Network 33
LD     V3.7
LD     Auto_Mode:V3.0
O      Single_Mode:V2019.7
ALD
A      Ini_OK_Tag:V0.7
A      DeviceIniOk:V0.6
LD     TS_ResetButton:V1000.0
EU
A      DeviceIniOk:V0.6
AN     IndexOrig_Pos:M9.0
O      Index_Motor:M25.0
OLD
AN     Index_Signal_Edge:V1000.7
AN     Reset_Button:M0.3
A      Fatal_Alarm:V107.7
AN     Station_Alarm:V107.6
=      Index_Motor:M25.0
Network 34
// M10.2 Servo Enable
LD     ServoEnable:M20.2
=      Q0.2
Network 35
LD     DelServoAlarm:M20.3
=      Q0.3
Network 36
LD     Up_Down_Cyl_1:M20.4
O      V2006.1
AN     Up_Down_Cyl_2:M20.5
=      Q0.4
Network 37
LD     Up_Down_Cyl_2:M20.5
O      V2006.0
AN     Up_Down_Cyl_1:M20.4
=      Q0.5
Network 38
LD     Pic_Product_Cyl_1:M20.6
O      V2006.2
=      Q0.6
Network 39
LD     Pic_Product_Cyl_2:M20.7
O      V2007.2
=      Q0.7
Network 40
LD     WaitStart:V3101.0
O      Running:V3101.1
AN     TW_R:M21.1
AN     TW_Buzzer:M21.2
=      TW_G:M21.0
Network 41
LD     Station_Alarm:V107.6
ON     Fatal_Alarm:V107.7
=      TW_R:M21.1
Network 42
LD     Maintain_mode:V2009.7
O      Product_set:V1999.7
=      TW_Buzzer:M21.2
Network 43
LD     TW_G:M21.0
=      Q1.0
Network 44
LD     TW_R:M21.1
=      Q1.1
Network 45
LD     TW_Buzzer:M21.2
=      Q1.2
Network 46
LD     Reset_lamp:M21.3
=      Q1.3
Network 47
LD     Bypass_Lamp:M21.4
=      Q1.4
Network 48 // 		
LD     M21.5
=      Q1.5
Network 49
LD     M21.6
=      Q1.6
Network 50
LD     M21.7
=      Q1.7
Network 51
LD     SV_3E_0:M22.0
=      Q2.0
Network 52
LD     SV_3E_1:M22.1
O      TS_Set_3E:V2001.0
=      Q2.1
Network 53
LD     SV_3F_0:M22.2
=      Q2.2
Network 54
LD     SV_3F_1:M22.3
O      TS_Set_3F:V2001.2
=      Q2.3
Network 55
LD     EnableTest_to_PC1:M22.4
O      TS_Current_Test:V2001.4
=      Q2.4
Network 56
LD     EnableTest_to_PC2:M22.5
O      V2001.6
=      Q2.5
Network 57
LD     M22.6
O      V2002.0
=      Q2.6
Network 58
LD     M22.7
O      V2002.2
=      Q2.7
Network 59
LD     SV_3A_0:M23.0
O      TS_Reset_3A:V2000.1
AN     TS_Set_3A:V2000.0
=      Q3.0
Network 60
LD     SV_3A_1:M23.1
O      TS_Set_3A:V2000.0
AN     TS_Reset_3A:V2000.1
=      Q3.1
Network 61
LD     SV_3B_0:M23.2
O      TS_Rset_3B0:V2000.3
=      Q3.2
Network 62
LD     SV_3B_1:M23.3
O      TS_Set_3B:V2000.2
=      Q3.3
Network 63
LD     SV_3C_0:M23.4
O      TS_Rset_3C_0:V2000.5
=      Q3.4
Network 64
LD     SV_3C_1:M23.5
O      TS_Set_3C:V2000.4
=      Q3.5
Network 65
LD     SV_3D_0:M23.6
O      TS_Rset_3D_0:V2000.7
=      Q3.6
Network 66
LD     SV_3D_1:M23.7
O      TS_Set_3D:V2000.6
=      Q3.7
Network 67
LD     SV_4A_0:M24.0
O      TS_Reset_4A:V2004.1
AN     TS_Set_4A:V2004.0
=      Q4.0
Network 68
LD     SV_4A_1:M24.1
O      TS_Set_4A:V2004.0
AN     TS_Reset_4A:V2004.1
=      Q4.1
Network 69
LD     SV_4B_2mmCYL:M24.2
O      V2004.2
=      Q4.2
Network 70
LD     SV_4C_RotateCyl:M24.3
O      V2004.4
=      Q4.3
Network 71
LD     SV_4D_RotateCyl:M24.4
O      V2004.6
=      Q4.4
Network 72
LD     Index_Brake:M24.5
LD     Safety_Curtain:M0.7
A      TS_IndexMotor:V1001.0
OLD
=      Q4.5
Network 73
LD     Servo_Brake:M24.6
=      Q4.6
Network 74
LD     MainValve:M24.7
=      Q4.7
Network 75
LD     Index_Motor:M25.0
LD     DeviceIniOk:V0.6
A      Safety_Curtain:M0.7
A      TS_IndexMotor:V1001.0
OLD
LPS
AN     TS_Stop:V1000.2
=      Q5.0
LPP
ED
R      Index_Signal_Edge:V1000.7, 1
Network 76
LD     ConverMotor:M25.1
AN     Maintain_mode:V2009.7
O      V1001.1
=      Q5.1
Network 77
LD     RejectBox_Cyl:M25.2
=      Q5.2
Network 78
LD     Start_Laser:M25.3
LD     Product_set:V1999.7
O      Maintain_mode:V2009.7
A      Sent_Ok:V50.7
OLD
=      Q5.3
Network 79
LD     Laser_done:M5.1
O      Stop_Laser:M25.4
O      Fatal_Alarm:V107.7
R      Sent_Ok:V50.7, 1
Network 80
LD     Stop_Laser:M25.4
O      TS_Laser_Stop:V2049.1
=      Q5.4
Network 81
LD     SpareM25_5:M25.5
=      Q5.5
Network 82
LD     Alarm1_ToPC:M25.6
=      Q5.6
Network 83
LD     Alarm2_ToPC:M25.7
=      Q5.7
Network 84
LD     StartLeakage_1:M26.0
O      V2005.0
AN     V2005.1
=      Q6.0
Network 85
LD     ResetLeakage_1:M26.1
O      V2005.1
AN     V2005.0
=      Q6.1
Network 86
LD     Romote_Eable_1:M26.2
=      Q6.2
Network 87
LD     M26.3
=      Q6.3
Network 88
LD     M26.4
=      Q6.4
Network 89
LD     M26.5
=      Q6.5
Network 90
LD     M26.6
=      Q6.6
Network 91
LD     M26.7
=      Q6.7
Network 92
LD     StartLeakage_2:M27.0
O      V2005.2
AN     V2005.3
=      Q7.0
Network 93
LD     ResetLeakage_2:M27.1
O      V2005.3
AN     V2005.2
=      Q7.1
Network 94
LD     Romote_Eable_2:M27.2
=      Q7.2
Network 95
LD     M27.3
=      Q7.3
Network 96
LD     M27.4
=      Q7.4
Network 97
LD     M27.5
=      Q7.5
Network 98
LD     M27.6
=      Q7.6
Network 99
LD     M27.7
O      V2007.7
=      Q7.7
END_SUBROUTINE_BLOCK

SUBROUTINE_BLOCK Tags:SBR14
TITLE=子程序注释
BEGIN
Network 1 // 网络标题
// 运行
LD     V2.7
O      StationRunTag:V0.0
AN     DeviceIniOk:V0.6
A      Fatal_Alarm:V107.7
AN     TS_Stop:V1000.2
=      StationRunTag:V0.0
Network 2
LD     V2.7
EU
MOVW   +0, VW2060
Network 3 // 网络标题
// 运行标志
LD     V2.2
O      V2.3
O      V2.4
O      V2.5
O      V2.6
AN     TS_ResetButton:V1000.0
AN     Station_Alarm:V107.6
A      Fatal_Alarm:V107.7
=      V2.7
A      Clock_1s:SM0.5
EU
+I     +1, VW2060
Network 4
LD     V26.1
O      V2.2
AN     V26.0
A      Fatal_Alarm:V107.7
=      V2.2
Network 5
LD     下行汽缸AB:V36.1
O      V2.3
AN     V36.0
AN     S3_Alarm:V138.7
A      Fatal_Alarm:V107.7
=      V2.3
Network 6
LDB<>  VB39, 0
=      Station3IniStatus:V1.3
Network 7
LD     V46.1
O      V2.4
AN     V46.0
AN     S4_Alarm:V148.7
A      Fatal_Alarm:V107.7
=      V2.4
Network 8
LDB<>  VB49, 0
=      Station4IniStatus:V1.4
Network 9
LD     V56.1
O      V2.5
AN     V56.0
AN     S5_Alarm:V158.7
A      Fatal_Alarm:V107.7
=      V2.5
Network 10
LDB<>  VB59, 0
=      Station5IniStatus:V1.5
Network 11
LD     V66.1
O      V2.6
AN     V66.0
AN     S6_Alarm:V168.7
A      Fatal_Alarm:V107.7
=      V2.6
Network 12
LDB<>  VB69, 0
=      Station6IniStatus:V1.6
Network 13
LD     Station3IniStatus:V1.3
O      Station4IniStatus:V1.4
O      Station5IniStatus:V1.5
O      Station6IniStatus:V1.6
=      IniTags:V1.7
Network 14
LD     DeviceIniOk:V0.6
LPS
A      Ini_OK_Tag:V0.7
=      SysIniOk:V0.5
LPP
AN     TS_ResetButton:V1000.0
AN     V2.7
=      V0.2
Network 15
LD     V0.2
EU
LD     Single_Mode:V2019.7
ED
OLD
MOVB   1, VB26
AENO
MOVB   1, VB36
AENO
MOVB   0, VB37
AENO
MOVB   1, VB46
AENO
MOVB   0, VB47
AENO
MOVB   1, VB56
AENO
MOVB   0, VB57
AENO
MOVB   1, VB66
AENO
MOVB   0, VB67
Network 16
// 硬件状态标志
LD     Cyl3A_S0:M3.0
A      Cyl3B_S0:M3.2
A      Cyl3C_S0:M3.4
A      Cyl2A_S0:M8.6
A      Cyl3D_S0:M3.6
A      Cyl3E_S0:M8.0
A      Cyl3F_S0:M8.2
A      Cyl_4A_S0:M4.0
A      Cyl3A_S0:M3.0
A      Cyl4B_S1:M4.3
A      Cyl4C_S0:M4.4
A      Cyl4D_S0:M4.6
AN     Laser_done:M5.1
A      Cyl6A_S0:M6.0
A      Cyl6B_S0:M6.2
A      Cyl6C_S0:M6.4
A      Servo_Home_Pos:M7.1
=      DeviceIniOk:V0.6
Network 17
// 系统初始状态标志
LDB=   VB26, 1
AB=    VB27, 0
AB=    VB36, 1
AB=    VB37, 0
AB=    VB46, 1
AB=    VB47, 0
AB=    VB56, 1
AB=    VB57, 0
AB=    VB66, 1
AB=    VB67, 0
AN     V123.7
AN     Station_Alarm:V107.6
A      Fatal_Alarm:V107.7
=      Ini_OK_Tag:V0.7
Network 18
LDB=   VB31, VB23
AB<>   VB31, 0
O      V2010.3
=      V30.1
Network 19
LDB=   VB32, VB23
AB<>   VB32, 0
O      V2010.3
=      V30.2
Network 20
LD     V30.1
O      V30.2
=      V30.3
Network 22
LDB=   VB41, 31
O      V40.4
O      V2010.4
=      S4_Product_Enable_Tag_1:V40.1
Network 23
LDB=   VB42, 31
O      V40.5
O      V2010.4
=      S4_Product_Enable_Tag_2:V40.2
Network 24
LD     S4_Product_Enable_Tag_1:V40.1
O      S4_Product_Enable_Tag_2:V40.2
AB<=   VB23, 4
=      S4_ProductEnable:V40.3
Network 25
LDB=   VB51, 32
O      V50.4
O      V2010.5
=      V50.1
Network 26
LDB=   VB52, 32
O      V50.5
O      V2010.5
=      V50.2
Network 27
LD     V50.1
O      V50.2
=      V50.3
Network 29
LDB<>  VB61, 0
=      V60.1
Network 30
LDB<>  VB62, 0
=      V60.2
Network 31
LD     V60.1
O      V60.2
=      V60.3
Network 32
LDB<   VB61, VB62
AB<>   VB61, 0
=      Release1st_1:V60.4
Network 33
LD     V66.1
O      V67.0
A      Release1st_1:V60.4
S      V1002.1, 1
Network 34
LD     V66.1
O      V67.0
A      Release1st_2:V60.5
S      V1002.2, 1
Network 35
LDB<   VB62, VB61
AB<>   VB62, 0
=      Release1st_2:V60.5
Network 36
LD     M31.1
O      M31.2
O      M31.3
O      M31.4
O      M31.5
=      V60.6
Network 37
LDB=   VB61, 34
OB=    VB62, 34
A      V60.3
AN     V360.2
AN     V360.3
AN     V360.4
AN     V360.5
=      V360.1
Network 38
LDB=   VB61, 21
OB=    VB62, 21
AN     V60.7
A      V60.3
=      V360.2
Network 39
LDB=   VB61, 22
OB=    VB62, 22
AN     V60.7
A      V60.3
AN     V360.2
=      V360.3
Network 40
LDB=   VB61, 23
OB=    VB62, 23
AN     V60.7
A      V60.3
AN     V360.2
AN     V360.3
=      V360.4
Network 41
LDB=   VB61, 29
OB=    VB62, 29
AN     V60.7
A      V60.3
AN     V360.2
AN     V360.3
AN     V360.4
=      V360.5
Network 42
LDN    DeviceIniOk:V0.6
AN     WaitStart:V3101.0
LD     SysIniOk:V0.5
AN     IndexOrig_Pos:M9.0
OLD
AN     Running:V3101.1
LD     Station_Alarm:V107.6
ON     Fatal_Alarm:V107.7
OLD
=      WaitIni:V3100.0
Network 43
LDN    DeviceIniOk:V0.6
AN     WaitStart:V3101.0
AN     Running:V3101.1
AN     WaitIni:V3100.0
=      Initilizing:V3100.1
Network 44
LD     SysIniOk:V0.5
AN     Running:V3101.1
AN     V121.6
A      IndexOrig_Pos:M9.0
=      WaitStart:V3101.0
Network 45
LD     StationRunTag:V0.0
O      TurnplateRunTag:V0.1
AN     Station_Alarm:V107.6
A      Fatal_Alarm:V107.7
=      Running:V3101.1
END_SUBROUTINE_BLOCK

SUBROUTINE_BLOCK PowerOn:SBR15
TITLE=子程序注释
BEGIN
Network 1
// 初始化语言为中文,自动模式
LD     First_Scan_On:SM0.1
O      Reset_Button:M0.3
O      TS_ResetButton:V1000.0
LPS
R      V1050.0, 1
S      Auto_Mode:V3.0, 1
R      Maintain_mode:V2009.7, 1
R      Single_Mode:V2019.7, 1
R      TS_IndexMotor:V1001.0, 1
R      V1002.1, 2
R      V3.7, 1
MOVD   +0, VD2000
AENO
MOVD   +0, VD2004
AENO
MOVW   +0, VW2008
LPP
MOVD   +0, VD2010
AENO
MOVD   +0, VD2014
AENO
MOVW   +0, VW2018
AENO
MOVW   +0, VW2020
AENO
MOVW   +4, VW2022
Network 2
LD     Station_Alarm:V107.6
ON     Fatal_Alarm:V107.7
R      V3.7, 1
Network 3 // 网络标题
// 网络注释
LD     First_Scan_On:SM0.1
MOVD   +0, VD0
AENO
MOVD   +0, VD4
Network 4
LD     First_Scan_On:SM0.1
MOVD   +0, VD10
AENO
MOVD   +0, VD14
Network 5
LD     First_Scan_On:SM0.1
MOVD   +0, VD24
Network 6
LD     First_Scan_On:SM0.1
MOVD   +0, VD24
AENO
MOVW   +0, VW28
Network 7
LD     First_Scan_On:SM0.1
MOVD   +0, VD34
AENO
MOVW   +0, VW38
Network 8
LD     First_Scan_On:SM0.1
MOVD   +0, VD44
AENO
MOVW   +0, VW48
Network 9
LD     First_Scan_On:SM0.1
MOVD   +0, VD54
AENO
MOVW   +0, VW58
Network 10
LD     First_Scan_On:SM0.1
MOVD   +0, VD64
AENO
MOVW   +0, VW68
AENO
MOVW   +0, VW63
END_SUBROUTINE_BLOCK

SUBROUTINE_BLOCK SyS_MSG:SBR16
TITLE=子程序注释
BEGIN
Network 1 // 网络标题
// vw106---vw168是系统报警信息（vw121是产品报警）
// vw176              是系统提示信息（包括待机、运行等信息）
LD     Always_On:SM0.0
LPS
MOVW   VW106, VW3106
AENO
MOVW   VW136, VW3136
AENO
MOVW   VW138, VW3138
LRD
MOVW   VW146, VW3146
AENO
MOVW   VW148, VW3148
LRD
MOVW   VW156, VW3156
AENO
MOVW   VW158, VW3158
LRD
MOVW   VW166, VW3166
AENO
MOVW   VW168, VW3168
LPP
MOVW   VW176, VW3176
AENO
MOVW   VW121, VW3121
AENO
MOVD   VD123, VD3123
END_SUBROUTINE_BLOCK

SUBROUTINE_BLOCK Communication_Laser:SBR18
TITLE=子程序注释
BEGIN
Network 1
LD     Always_On:SM0.0
MOVB   'S', VB4050
AENO
MOVB   'T', VB4051
AENO
MOVB   'E', VB4098
AENO
MOVB   'D', VB4099
Network 2
LD     Always_On:SM0.0
MOVB   'S', VB4000
AENO
MOVB   'T', VB4001
AENO
MOVB   'E', VB4048
AENO
MOVB   'D', VB4049
END_SUBROUTINE_BLOCK

SUBROUTINE_BLOCK TypeCheck:SBR19
TITLE=子程序注释
BEGIN
Network 1
LDN    S1_Cover_Group:M1.4
AN     S1_OE1:M1.1
AN     S1_OE2:M1.2
AN     S1_OE3:M1.3
AN     S1_Ball_Screw:M1.0
MOVB   0, VB21
Network 2 // 网络标题
// vb=0, 未检测到产品
LD     S1_Cover_Group:M1.4
AN     S1_OE1:M1.1
AN     S1_OE2:M1.2
AN     S1_OE3:M1.3
LD     S1_ORing:M1.6
A      S1_Ball_Screw:M1.0
O      Always_On:SM0.0
ALD
MOVB   1, VB21
Network 3
// vb=2, Type=007 878-20
LD     S1_Cover_Group:M1.4
A      S1_OE1:M1.1
AN     S1_OE2:M1.2
AN     S1_OE3:M1.3
LD     S1_ORing:M1.6
A      S1_Ball_Screw:M1.0
O      Always_On:SM0.0
ALD
MOVB   2, VB21
Network 4
// vb=3, Type=007 878-21
LD     S1_Cover_Group:M1.4
AN     S1_OE1:M1.1
A      S1_OE2:M1.2
AN     S1_OE3:M1.3
LD     S1_ORing:M1.6
A      S1_Ball_Screw:M1.0
O      Always_On:SM0.0
ALD
MOVB   3, VB21
Network 5
// vb=4,Type=007 878-22
LD     S1_Cover_Group:M1.4
AN     S1_OE1:M1.1
AN     S1_OE2:M1.2
A      S1_OE3:M1.3
LD     S1_ORing:M1.6
A      S1_Ball_Screw:M1.0
O      Always_On:SM0.0
ALD
MOVB   4, VB21
Network 6
// vb=5,Type=007 878-00
LDN    S1_Cover_Group:M1.4
A      S1_Color:M1.5
AN     S1_OE1:M1.1
AN     S1_OE2:M1.2
AN     S1_OE3:M1.3
LD     S1_ORing:M1.6
O      Always_On:SM0.0
ALD
A      S1_Ball_Screw:M1.0
MOVB   5, VB21
Network 7
// vb=6,Type=007 878-04
LDN    S1_Cover_Group:M1.4
AN     S1_Color:M1.5
AN     S1_OE1:M1.1
AN     S1_OE2:M1.2
AN     S1_OE3:M1.3
LD     S1_ORing:M1.6
O      Always_On:SM0.0
ALD
A      S1_Ball_Screw:M1.0
MOVB   6, VB21
Network 8 // 网络标题
// 网络注释
END_SUBROUTINE_BLOCK

SUBROUTINE_BLOCK TypeCheck1:SBR20
TITLE=
BEGIN
Network 1
LDN    S2_Cover_Group:M2.4
AN     S2OE21:M2.1
AN     S2OE2:M2.2
AN     S2OE3:M2.3
AN     S2ORing:M2.6
AN     S2Ball_Screw:M2.0
MOVB   0, VB22
Network 2 // 网络标题
// vb=0, 未检测到产品
LD     S2_Cover_Group:M2.4
AN     S2OE21:M2.1
AN     S2OE2:M2.2
AN     S2OE3:M2.3
LD     S2ORing:M2.6
A      S2Ball_Screw:M2.0
O      Always_On:SM0.0
ALD
MOVB   1, VB22
Network 3
// vb=2, Type=007 878-20
LD     S2_Cover_Group:M2.4
A      S2OE21:M2.1
AN     S2OE2:M2.2
AN     S2OE3:M2.3
LD     S2ORing:M2.6
A      S2Ball_Screw:M2.0
O      Always_On:SM0.0
ALD
MOVB   2, VB22
Network 4
// vb=3, Type=007 878-21
LD     S2_Cover_Group:M2.4
AN     S2OE21:M2.1
A      S2OE2:M2.2
AN     S2OE3:M2.3
LD     S2ORing:M2.6
A      S2Ball_Screw:M2.0
O      Always_On:SM0.0
ALD
MOVB   3, VB22
Network 5
// vb=4,Type=007 878-22
LD     S2_Cover_Group:M2.4
AN     S2OE21:M2.1
AN     S2OE2:M2.2
A      S2OE3:M2.3
LD     S2_Cover_Group:M2.4
A      S2Ball_Screw:M2.0
O      Always_On:SM0.0
ALD
MOVB   4, VB22
Network 6
// vb=5,Type=007 878-00
LDN    S2_Cover_Group:M2.4
A      Color_Sensor:M2.5
AN     S2OE21:M2.1
AN     S2OE2:M2.2
AN     S2OE3:M2.3
LD     S2ORing:M2.6
O      Always_On:SM0.0
ALD
A      S2Ball_Screw:M2.0
MOVB   5, VB22
Network 7
// vb=6,Type=007 878-04
LDN    S2_Cover_Group:M2.4
AN     Color_Sensor:M2.5
AN     S2OE21:M2.1
AN     S2OE2:M2.2
AN     S2OE3:M2.3
LD     S2ORing:M2.6
O      Always_On:SM0.0
ALD
A      S2Ball_Screw:M2.0
MOVB   6, VB22
Network 8 // 网络标题
// 网络注释
END_SUBROUTINE_BLOCK

INTERRUPT_BLOCK Orig_Pos:INT0
TITLE=中断程序注释
BEGIN
Network 1 // 网络标题
// 网络注释
LD     Always_On:SM0.0
S      M31.0, 1
END_INTERRUPT_BLOCK

INTERRUPT_BLOCK Current_NG:INT1
TITLE=中断程序注释
BEGIN
Network 1 // 网络标题
// 网络注释
LD     Always_On:SM0.0
S      M31.1, 1
Network 2 // 网络标题
// 网络注释
END_INTERRUPT_BLOCK

INTERRUPT_BLOCK RunTime_NG:INT2
TITLE=中断程序注释
BEGIN
Network 1 // 网络标题
// 网络注释
LD     Always_On:SM0.0
S      M31.2, 1
Network 2 // 网络标题
// 网络注释
END_INTERRUPT_BLOCK

INTERRUPT_BLOCK LKG_NG:INT3
TITLE=中断程序注释
BEGIN
Network 1 // 网络标题
// 网络注释
LD     Always_On:SM0.0
S      M31.3, 1
Network 2 // 网络标题
// 网络注释
END_INTERRUPT_BLOCK

INTERRUPT_BLOCK NoTest:INT4
TITLE=中断程序注释
BEGIN
Network 1 // 网络标题
// 网络注释
LD     Always_On:SM0.0
S      M31.4, 1
Network 2 // 网络标题
// 网络注释
END_INTERRUPT_BLOCK

INTERRUPT_BLOCK OK_Pos:INT5
TITLE=中断程序注释
BEGIN
Network 1 // 网络标题
// 网络注释
LD     Always_On:SM0.0
S      M31.5, 1
R      M31.4, 1
Network 2 // 网络标题
// 网络注释
END_INTERRUPT_BLOCK

INTERRUPT_BLOCK Servo_Ini:INT6
TITLE=中断程序注释
BEGIN
Network 1 // 网络标题
// 网络注释
LD     V69.3
S      V31.6, 1
Network 2 // 网络标题
// 网络注释
LD     V69.4
S      V31.7, 1
END_INTERRUPT_BLOCK
